LIN {X 0,Y 523.947,Z 221.718,A -85,B 0,C 180,E1 -4737.68,E2 -4737.68} C_VEL
LIN {X 0,Y 523.963,Z 221.716,A -85,B 0,C 180,E1 -4740.677,E2 -4740.677} C_VEL
LIN {X 0,Y 523.944,Z 221.72,A -85,B 0,C 180,E1 -4743.726,E2 -4743.726} C_VEL
LIN {X 0,Y 523.98,Z 221.866,A -85,B 0,C 180,E1 -4746.586,E2 -4746.586} C_VEL
LIN {X 0,Y 525.206,Z 229.619,A -85,B 0,C 180,E1 -4747.994,E2 -4747.994} C_VEL
LIN {X 0,Y 524.786,Z 247.778,A -85,B 0,C 180,E1 -4751.048,E2 -4751.048} C_VEL
LIN {X 0,Y 524.374,Z 265.93,A -85,B 0,C 180,E1 -4754.052,E2 -4754.052} C_VEL
LIN {X 0,Y 524.311,Z 270.834,A -85,B 0,C 180,E1 -4754.823,E2 -4754.823} C_VEL
LIN {X 0,Y 525.641,Z 279.389,A -85,B 0,C 180,E1 -4755.009,E2 -4755.009} C_VEL
LIN {X 0,Y 525.957,Z 285.477,A -85,B 0,C 180,E1 -4755.103,E2 -4755.103} C_VEL
LIN {X 0,Y 525.554,Z 378.201,A -85,B 0,C 180,E1 -4756.391,E2 -4756.391} C_VEL
LIN {X 0,Y 525.355,Z 391.598,A -85,B 0,C 180,E1 -4756.731,E2 -4756.731} C_VEL
LIN {X 0,Y 525.029,Z 404.942,A -85,B 0,C 180,E1 -4757.239,E2 -4757.239} C_VEL
LIN {X 0,Y 524.818,Z 416.473,A -85,B 0,C 180,E1 -4757.844,E2 -4757.844} C_VEL
LIN {X 0,Y 524.548,Z 427.744,A -85,B 0,C 180,E1 -4758.601,E2 -4758.601} C_VEL
LIN {X 0,Y 524.212,Z 438.191,A -85,B 0,C 180,E1 -4759.474,E2 -4759.474} C_VEL
LIN {X 0,Y 524.028,Z 446.732,A -85,B 0,C 180,E1 -4760.348,E2 -4760.348} C_VEL
LIN {X 0,Y 523.819,Z 454.609,A -85,B 0,C 180,E1 -4761.317,E2 -4761.317} C_VEL
LIN {X 0,Y 523.624,Z 462.299,A -85,B 0,C 180,E1 -4762.479,E2 -4762.479} C_VEL
LIN {X 0,Y 523.496,Z 469.383,A -85,B 0,C 180,E1 -4763.833,E2 -4763.833} C_VEL
LIN {X 0,Y 523.385,Z 474.095,A -85,B 0,C 180,E1 -4764.992,E2 -4764.992} C_VEL
LIN {X 0,Y 523.445,Z 477.695,A -85,B 0,C 180,E1 -4766.15,E2 -4766.15} C_VEL
LIN {X 0,Y 523.369,Z 479.552,A -85,B 0,C 180,E1 -4766.92,E2 -4766.92} C_VEL
LIN {X 0,Y 523.335,Z 480.943,A -85,B 0,C 180,E1 -4767.69,E2 -4767.69} C_VEL
LIN {X 0,Y 523.25,Z 482.542,A -85,B 0,C 180,E1 -4769.229,E2 -4769.229} C_VEL
LIN {X 0,Y 523.247,Z 482.758,A -85,B 0,C 180,E1 -4769.999,E2 -4769.999} C_VEL
LIN {X 0,Y 523.275,Z 481.938,A -85,B 0,C 180,E1 -4771.538,E2 -4771.538} C_VEL
LIN {X 0,Y 523.335,Z 480.947,A -85,B 0,C 180,E1 -4772.308,E2 -4772.308} C_VEL
LIN {X 0,Y 523.368,Z 479.556,A -85,B 0,C 180,E1 -4773.078,E2 -4773.078} C_VEL
LIN {X 0,Y 523.424,Z 476.63,A -85,B 0,C 180,E1 -4774.234,E2 -4774.234} C_VEL
LIN {X 0,Y 523.462,Z 472.668,A -85,B 0,C 180,E1 -4775.391,E2 -4775.391} C_VEL
LIN {X 0,Y 523.503,Z 466.604,A -85,B 0,C 180,E1 -4776.738,E2 -4776.738} C_VEL
LIN {X 0,Y 523.674,Z 459.908,A -85,B 0,C 180,E1 -4777.905,E2 -4777.905} C_VEL
LIN {X 0,Y 523.861,Z 451.635,A -85,B 0,C 180,E1 -4779.068,E2 -4779.068} C_VEL
LIN {X 0,Y 524.081,Z 443.153,A -85,B 0,C 180,E1 -4780.038,E2 -4780.038} C_VEL
LIN {X 0,Y 524.365,Z 432.668,A -85,B 0,C 180,E1 -4781.009,E2 -4781.009} C_VEL
LIN {X 0,Y 524.659,Z 421.21,A -85,B 0,C 180,E1 -4781.86,E2 -4781.86} C_VEL
LIN {X 0,Y 524.974,Z 408.979,A -85,B 0,C 180,E1 -4782.563,E2 -4782.563} C_VEL
LIN {X 0,Y 525.247,Z 396.61,A -85,B 0,C 180,E1 -4783.097,E2 -4783.097} C_VEL
LIN {X 0,Y 525.41,Z 383.894,A -85,B 0,C 180,E1 -4783.487,E2 -4783.487} C_VEL
LIN {X 0,Y 525.622,Z 368.754,A -85,B 0,C 180,E1 -4783.752,E2 -4783.752} C_VEL
LIN {X 0,Y 525.857,Z 280.922,A -85,B 0,C 180,E1 -4784.963,E2 -4784.963} C_VEL
LIN {X 0,Y 524.29,Z 270.905,A -85,B 0,C 180,E1 -4785.169,E2 -4785.169} C_VEL
LIN {X 0,Y 524.336,Z 265.85,A -85,B 0,C 180,E1 -4785.947,E2 -4785.947} C_VEL
LIN {X 0,Y 524.686,Z 248.802,A -85,B 0,C 180,E1 -4788.751,E2 -4788.751} C_VEL
LIN {X 0,Y 525.189,Z 230.523,A -85,B 0,C 180,E1 -4791.797,E2 -4791.797} C_VEL
LIN {X 0,Y 524.722,Z 225.824,A -85,B 0,C 180,E1 -4792.615,E2 -4792.615} C_VEL
LIN {X 0,Y 523.962,Z 221.786,A -85,B 0,C 180,E1 -4793.386,E2 -4793.386} C_VEL
LIN {X 0,Y 523.944,Z 221.72,A -85,B 0,C 180,E1 -4796.272,E2 -4796.272} C_VEL
LIN {X 0,Y 523.931,Z 221.717,A -85,B 0,C 180,E1 -4798.874,E2 -4798.874} C_VEL
LIN {X 0,Y 523.921,Z 221.723,A -85,B 0,C 180,E1 -4801.542,E2 -4801.542} C_VEL
LIN {X 0,Y 523.932,Z 221.72,A -85,B 0,C 180,E1 -4804.288,E2 -4804.288} C_VEL
LIN {X 0,Y 523.904,Z 221.721,A -85,B 0,C 180,E1 -4807.131,E2 -4807.131} C_VEL
LIN {X 0,Y 523.938,Z 221.725,A -85,B 0,C 180,E1 -4810.128,E2 -4810.128} C_VEL
LIN {X 0,Y 523.922,Z 221.723,A -85,B 0,C 180,E1 -4812.455,E2 -4812.455} C_VEL
LIN {X 0,Y 523.94,Z 221.715,A -85,B 0,C 180,E1 -4815.308,E2 -4815.308} C_VEL
LIN {X 0,Y 523.938,Z 221.721,A -85,B 0,C 180,E1 -4818.69,E2 -4818.69} C_VEL
LIN {X 0,Y 523.909,Z 221.721,A -85,B 0,C 180,E1 -4821.896,E2 -4821.896} C_VEL
LIN {X 0,Y 523.919,Z 221.722,A -85,B 0,C 180,E1 -4824.909,E2 -4824.909} C_VEL
LIN {X 0,Y 523.93,Z 221.715,A -85,B 0,C 180,E1 -4827.678,E2 -4827.678} C_VEL
LIN {X 0,Y 523.946,Z 221.722,A -85,B 0,C 180,E1 -4830.675,E2 -4830.675} C_VEL
LIN {X 0,Y 523.898,Z 221.72,A -85,B 0,C 180,E1 -4833.722,E2 -4833.722} C_VEL
LIN {X 0,Y 523.9,Z 221.721,A -85,B 0,C 180,E1 -4836.267,E2 -4836.267} C_VEL
LIN {X 0,Y 523.935,Z 221.722,A -85,B 0,C 180,E1 -4838.764,E2 -4838.764} C_VEL
LIN {X 0,Y 523.928,Z 221.723,A -85,B 0,C 180,E1 -4841.217,E2 -4841.217} C_VEL
LIN {X 0,Y 523.899,Z 221.721,A -85,B 0,C 180,E1 -4843.635,E2 -4843.635} C_VEL
LIN {X 0,Y 523.902,Z 221.72,A -85,B 0,C 180,E1 -4846.024,E2 -4846.024} C_VEL
LIN {X 0,Y 524.003,Z 221.705,A -85,B 0,C 180,E1 -4848.391,E2 -4848.391} C_VEL
LIN {X 0,Y 523.934,Z 221.719,A -85,B 0,C 180,E1 -4851.512,E2 -4851.512} C_VEL
LIN {X 0,Y 523.997,Z 221.711,A -85,B 0,C 180,E1 -4853.838,E2 -4853.838} C_VEL
LIN {X 0,Y 523.934,Z 221.725,A -85,B 0,C 180,E1 -4855.381,E2 -4855.381} C_VEL
LIN {X 0,Y 524.082,Z 221.703,A -85,B 0,C 180,E1 -4857.691,E2 -4857.691} C_VEL
LIN {X 0,Y 524.071,Z 221.7,A -85,B 0,C 180,E1 -4859.997,E2 -4859.997} C_VEL
LIN {X 0,Y 524.079,Z 221.698,A -85,B 0,C 180,E1 -4862.303,E2 -4862.303} C_VEL
LIN {X 0,Y 523.982,Z 221.713,A -85,B 0,C 180,E1 -4866.157,E2 -4866.157} C_VEL
LIN {X 0,Y 523.96,Z 221.714,A -85,B 0,C 180,E1 -4869.259,E2 -4869.259} C_VEL
LIN {X 0,Y 523.977,Z 221.719,A -85,B 0,C 180,E1 -4871.734,E2 -4871.734} C_VEL
LIN {X 0,Y 523.963,Z 221.713,A -85,B 0,C 180,E1 -4875.046,E2 -4875.046} C_VEL
LIN {X 0,Y 523.92,Z 221.726,A -85,B 0,C 180,E1 -4877.967,E2 -4877.967} C_VEL
LIN {X 0,Y 523.946,Z 221.72,A -85,B 0,C 180,E1 -4880.407,E2 -4880.407} C_VEL
LIN {X 0,Y 523.884,Z 221.723,A -85,B 0,C 180,E1 -4882.891,E2 -4882.891} C_VEL
LIN {X 0,Y 523.954,Z 221.719,A -85,B 0,C 180,E1 -4886.016,E2 -4886.016} C_VEL
LIN {X 0,Y 523.908,Z 221.72,A -85,B 0,C 180,E1 -4888.872,E2 -4888.872} C_VEL
LIN {X 0,Y 523.891,Z 221.722,A -85,B 0,C 180,E1 -4891.541,E2 -4891.541} C_VEL
LIN {X 0,Y 523.912,Z 221.726,A -85,B 0,C 180,E1 -4894.287,E2 -4894.287} C_VEL
LIN {X 0,Y 523.879,Z 221.726,A -85,B 0,C 180,E1 -4897.129,E2 -4897.129} C_VEL
LIN {X 0,Y 523.932,Z 221.72,A -85,B 0,C 180,E1 -4900.132,E2 -4900.132} C_VEL
LIN {X 0,Y 523.908,Z 221.726,A -85,B 0,C 180,E1 -4902.458,E2 -4902.458} C_VEL
LIN {X 0,Y 523.917,Z 221.724,A -85,B 0,C 180,E1 -4905.306,E2 -4905.306} C_VEL
LIN {X 0,Y 523.893,Z 221.73,A -85,B 0,C 180,E1 -4906.862,E2 -4906.862} C_VEL
LIN {X 0,Y 523.611,Z 222.17,A -85,B 0,C 180,E1 -4907.286,E2 -4907.286} C_VEL
LIN {X 0,Y 522.901,Z 223.307,A -85,B 0,C 180,E1 -4907.69,E2 -4907.69} C_VEL
LIN {X 0,Y 520.809,Z 226.879,A -85,B 0,C 180,E1 -4908.44,E2 -4908.44} C_VEL
LIN {X 0,Y 518.658,Z 231.406,A -85,B 0,C 180,E1 -4909.162,E2 -4909.162} C_VEL
LIN {X 0,Y 517.705,Z 234.729,A -85,B 0,C 180,E1 -4909.714,E2 -4909.714} C_VEL
LIN {X 0,Y 517.612,Z 235.807,A -85,B 0,C 180,E1 -4909.904,E2 -4909.904} C_VEL
LIN {X 0,Y 517.285,Z 252.208,A -85,B 0,C 180,E1 -4912.803,E2 -4912.803} C_VEL
LIN {X 0,Y 517.261,Z 257.358,A -85,B 0,C 180,E1 -4913.666,E2 -4913.666} C_VEL
LIN {X 0,Y 519.08,Z 267.962,A -85,B 0,C 180,E1 -4913.896,E2 -4913.896} C_VEL
LIN {X 0,Y 518.62,Z 364.773,A -85,B 0,C 180,E1 -4915.266,E2 -4915.266} C_VEL
LIN {X 0,Y 518.388,Z 378.478,A -85,B 0,C 180,E1 -4915.628,E2 -4915.628} C_VEL
LIN {X 0,Y 518.17,Z 391.423,A -85,B 0,C 180,E1 -4916.141,E2 -4916.141} C_VEL
LIN {X 0,Y 517.873,Z 403.178,A -85,B 0,C 180,E1 -4916.777,E2 -4916.777} C_VEL
LIN {X 0,Y 517.535,Z 414.859,A -85,B 0,C 180,E1 -4917.588,E2 -4917.588} C_VEL
LIN {X 0,Y 517.253,Z 424.904,A -85,B 0,C 180,E1 -4918.461,E2 -4918.461} C_VEL
LIN {X 0,Y 516.989,Z 433.313,A -85,B 0,C 180,E1 -4919.353,E2 -4919.353} C_VEL
LIN {X 0,Y 516.714,Z 442.175,A -85,B 0,C 180,E1 -4920.505,E2 -4920.505} C_VEL
LIN {X 0,Y 516.594,Z 448.832,A -85,B 0,C 180,E1 -4921.567,E2 -4921.567} C_VEL
LIN {X 0,Y 516.445,Z 455.453,A -85,B 0,C 180,E1 -4922.88,E2 -4922.88} C_VEL
LIN {X 0,Y 516.342,Z 460.483,A -85,B 0,C 180,E1 -4924.181,E2 -4924.181} C_VEL
LIN {X 0,Y 516.281,Z 463.056,A -85,B 0,C 180,E1 -4925.041,E2 -4925.041} C_VEL
LIN {X 0,Y 516.233,Z 465.12,A -85,B 0,C 180,E1 -4925.896,E2 -4925.896} C_VEL
LIN {X 0,Y 516.168,Z 466.619,A -85,B 0,C 180,E1 -4926.745,E2 -4926.745} C_VEL
LIN {X 0,Y 516.15,Z 467.852,A -85,B 0,C 180,E1 -4927.791,E2 -4927.791} C_VEL
LIN {X 0,Y 516.16,Z 468.321,A -85,B 0,C 180,E1 -4929.268,E2 -4929.268} C_VEL
LIN {X 0,Y 516.202,Z 467.974,A -85,B 0,C 180,E1 -4930.102,E2 -4930.102} C_VEL
LIN {X 0,Y 516.163,Z 467.205,A -85,B 0,C 180,E1 -4930.928,E2 -4930.928} C_VEL
LIN {X 0,Y 516.222,Z 464.765,A -85,B 0,C 180,E1 -4932.347,E2 -4932.347} C_VEL
LIN {X 0,Y 516.313,Z 460.827,A -85,B 0,C 180,E1 -4933.798,E2 -4933.798} C_VEL
LIN {X 0,Y 516.425,Z 456.142,A -85,B 0,C 180,E1 -4935.048,E2 -4935.048} C_VEL
LIN {X 0,Y 516.564,Z 449.361,A -85,B 0,C 180,E1 -4936.428,E2 -4936.428} C_VEL
LIN {X 0,Y 516.761,Z 441.828,A -85,B 0,C 180,E1 -4937.633,E2 -4937.633} C_VEL
LIN {X 0,Y 516.945,Z 434.081,A -85,B 0,C 180,E1 -4938.643,E2 -4938.643} C_VEL
LIN {X 0,Y 517.271,Z 424.866,A -85,B 0,C 180,E1 -4939.63,E2 -4939.63} C_VEL
LIN {X 0,Y 517.531,Z 414.551,A -85,B 0,C 180,E1 -4940.524,E2 -4940.524} C_VEL
LIN {X 0,Y 517.896,Z 403.064,A -85,B 0,C 180,E1 -4941.318,E2 -4941.318} C_VEL
LIN {X 0,Y 518.131,Z 391.865,A -85,B 0,C 180,E1 -4941.927,E2 -4941.927} C_VEL
LIN {X 0,Y 518.4,Z 379.448,A -85,B 0,C 180,E1 -4942.43,E2 -4942.43} C_VEL
LIN {X 0,Y 518.63,Z 366.936,A -85,B 0,C 180,E1 -4942.776,E2 -4942.776} C_VEL
LIN {X 0,Y 518.731,Z 346.658,A -85,B 0,C 180,E1 -4943.095,E2 -4943.095} C_VEL
LIN {X 0,Y 518.965,Z 267.136,A -85,B 0,C 180,E1 -4944.208,E2 -4944.208} C_VEL
LIN {X 0,Y 517.256,Z 257.525,A -85,B 0,C 180,E1 -4944.421,E2 -4944.421} C_VEL
LIN {X 0,Y 517.473,Z 246.928,A -85,B 0,C 180,E1 -4946.302,E2 -4946.302} C_VEL
LIN {X 0,Y 517.903,Z 232.103,A -85,B 0,C 180,E1 -4949.029,E2 -4949.029} C_VEL
LIN {X 0,Y 517.75,Z 226.931,A -85,B 0,C 180,E1 -4950.001,E2 -4950.001} C_VEL
LIN {X 0,Y 517.036,Z 222.663,A -85,B 0,C 180,E1 -4950.877,E2 -4950.877} C_VEL
LIN {X 0,Y 516.976,Z 222.591,A -85,B 0,C 180,E1 -4953.118,E2 -4953.118} C_VEL
LIN {X 0,Y 516.961,Z 222.586,A -85,B 0,C 180,E1 -4956.245,E2 -4956.245} C_VEL
LIN {X 0,Y 516.909,Z 222.598,A -85,B 0,C 180,E1 -4959.391,E2 -4959.391} C_VEL
LIN {X 0,Y 516.941,Z 222.593,A -85,B 0,C 180,E1 -4961.826,E2 -4961.826} C_VEL
LIN {X 0,Y 516.901,Z 222.593,A -85,B 0,C 180,E1 -4965.148,E2 -4965.148} C_VEL
LIN {X 0,Y 516.884,Z 222.597,A -85,B 0,C 180,E1 -4968.225,E2 -4968.225} C_VEL
LIN {X 0,Y 516.873,Z 222.595,A -85,B 0,C 180,E1 -4970.704,E2 -4970.704} C_VEL
LIN {X 0,Y 516.851,Z 222.607,A -85,B 0,C 180,E1 -4974.076,E2 -4974.076} C_VEL
LIN {X 0,Y 516.851,Z 222.6,A -85,B 0,C 180,E1 -4976.663,E2 -4976.663} C_VEL
LIN {X 0,Y 516.875,Z 222.596,A -85,B 0,C 180,E1 -4979.527,E2 -4979.527} C_VEL
LIN {X 0,Y 516.861,Z 222.602,A -85,B 0,C 180,E1 -4982.546,E2 -4982.546} C_VEL
LIN {X 0,Y 516.821,Z 222.601,A -85,B 0,C 180,E1 -4985.331,E2 -4985.331} C_VEL
LIN {X 0,Y 516.843,Z 222.605,A -85,B 0,C 180,E1 -4988.72,E2 -4988.72} C_VEL
LIN {X 0,Y 516.854,Z 222.598,A -85,B 0,C 180,E1 -4991.782,E2 -4991.782} C_VEL
LIN {X 0,Y 516.871,Z 222.6,A -85,B 0,C 180,E1 -4995.011,E2 -4995.011} C_VEL
LIN {X 0,Y 516.865,Z 222.6,A -85,B 0,C 180,E1 -4998.406,E2 -4998.406} C_VEL
LIN {X 0,Y 516.856,Z 222.601,A -85,B 0,C 180,E1 -5001.288,E2 -5001.288} C_VEL
LIN {X 0,Y 516.853,Z 222.598,A -85,B 0,C 180,E1 -5004.224,E2 -5004.224} C_VEL
LIN {X 0,Y 516.864,Z 222.606,A -85,B 0,C 180,E1 -5007.056,E2 -5007.056} C_VEL
LIN {X 0,Y 516.849,Z 222.599,A -85,B 0,C 180,E1 -5009.798,E2 -5009.798} C_VEL
LIN {X 0,Y 516.861,Z 222.597,A -85,B 0,C 180,E1 -5012.468,E2 -5012.468} C_VEL
LIN {X 0,Y 516.861,Z 222.602,A -85,B 0,C 180,E1 -5015.65,E2 -5015.65} C_VEL
LIN {X 0,Y 516.878,Z 222.594,A -85,B 0,C 180,E1 -5018.466,E2 -5018.466} C_VEL
LIN {X 0,Y 516.884,Z 222.595,A -85,B 0,C 180,E1 -5020.958,E2 -5020.958} C_VEL
LIN {X 0,Y 516.878,Z 222.601,A -85,B 0,C 180,E1 -5023.413,E2 -5023.413} C_VEL
LIN {X 0,Y 516.879,Z 222.602,A -85,B 0,C 180,E1 -5025.837,E2 -5025.837} C_VEL
LIN {X 0,Y 516.926,Z 222.591,A -85,B 0,C 180,E1 -5028.236,E2 -5028.236} C_VEL
LIN {X 0,Y 516.93,Z 222.591,A -85,B 0,C 180,E1 -5031.402,E2 -5031.402} C_VEL
LIN {X 0,Y 516.983,Z 222.583,A -85,B 0,C 180,E1 -5034.543,E2 -5034.543} C_VEL
LIN {X 0,Y 517.075,Z 222.573,A -85,B 0,C 180,E1 -5037.666,E2 -5037.666} C_VEL
LIN {X 0,Y 517.072,Z 222.572,A -85,B 0,C 180,E1 -5040.782,E2 -5040.782} C_VEL
LIN {X 0,Y 516.949,Z 222.586,A -85,B 0,C 180,E1 -5043.12,E2 -5043.12} C_VEL
LIN {X 0,Y 516.978,Z 222.59,A -85,B 0,C 180,E1 -5046.246,E2 -5046.246} C_VEL
LIN {X 0,Y 516.918,Z 222.589,A -85,B 0,C 180,E1 -5049.393,E2 -5049.393} C_VEL
LIN {X 0,Y 516.964,Z 222.584,A -85,B 0,C 180,E1 -5051.809,E2 -5051.809} C_VEL
LIN {X 0,Y 516.949,Z 222.588,A -85,B 0,C 180,E1 -5055.145,E2 -5055.145} C_VEL
LIN {X 0,Y 516.923,Z 222.591,A -85,B 0,C 180,E1 -5058.225,E2 -5058.225} C_VEL
LIN {X 0,Y 516.914,Z 222.598,A -85,B 0,C 180,E1 -5060.704,E2 -5060.704} C_VEL
LIN {X 0,Y 516.869,Z 222.6,A -85,B 0,C 180,E1 -5063.226,E2 -5063.226} C_VEL
LIN {X 0,Y 516.895,Z 222.592,A -85,B 0,C 180,E1 -5066.183,E2 -5066.183} C_VEL
LIN {X 0,Y 516.917,Z 222.596,A -85,B 0,C 180,E1 -5069.307,E2 -5069.307} C_VEL
LIN {X 0,Y 516.905,Z 222.592,A -85,B 0,C 180,E1 -5072.543,E2 -5072.543} C_VEL
LIN {X 0,Y 516.868,Z 222.606,A -85,B 0,C 180,E1 -5075.328,E2 -5075.328} C_VEL
LIN {X 0,Y 516.891,Z 222.595,A -85,B 0,C 180,E1 -5077.943,E2 -5077.943} C_VEL
LIN {X 0,Y 516.866,Z 222.596,A -85,B 0,C 180,E1 -5080.745,E2 -5080.745} C_VEL
LIN {X 0,Y 516.894,Z 222.597,A -85,B 0,C 180,E1 -5083.904,E2 -5083.904} C_VEL
LIN {X 0,Y 516.893,Z 222.596,A -85,B 0,C 180,E1 -5086.108,E2 -5086.108} C_VEL
LIN {X 0,Y 516.865,Z 222.598,A -85,B 0,C 180,E1 -5089.255,E2 -5089.255} C_VEL
LIN {X 0,Y 516.873,Z 222.599,A -85,B 0,C 180,E1 -5092.274,E2 -5092.274} C_VEL
LIN {X 0,Y 516.892,Z 222.593,A -85,B 0,C 180,E1 -5095.175,E2 -5095.175} C_VEL
LIN {X 0,Y 516.885,Z 222.602,A -85,B 0,C 180,E1 -5097.975,E2 -5097.975} C_VEL
LIN {X 0,Y 516.931,Z 222.592,A -85,B 0,C 180,E1 -5100.695,E2 -5100.695} C_VEL
LIN {X 0,Y 516.909,Z 222.597,A -85,B 0,C 180,E1 -5103.814,E2 -5103.814} C_VEL
LIN {X 0,Y 516.941,Z 222.705,A -85,B 0,C 180,E1 -5106.407,E2 -5106.407} C_VEL
LIN {X 0,Y 518.254,Z 230.732,A -85,B 0,C 180,E1 -5107.893,E2 -5107.893} C_VEL
LIN {X 0,Y 517.84,Z 247.689,A -85,B 0,C 180,E1 -5110.784,E2 -5110.784} C_VEL
LIN {X 0,Y 517.378,Z 265.836,A -85,B 0,C 180,E1 -5113.83,E2 -5113.83} C_VEL
LIN {X 0,Y 517.302,Z 270.899,A -85,B 0,C 180,E1 -5114.622,E2 -5114.622} C_VEL
LIN {X 0,Y 519.108,Z 283.14,A -85,B 0,C 180,E1 -5114.87,E2 -5114.87} C_VEL
LIN {X 0,Y 518.659,Z 378.034,A -85,B 0,C 180,E1 -5116.207,E2 -5116.207} C_VEL
LIN {X 0,Y 518.443,Z 391.457,A -85,B 0,C 180,E1 -5116.55,E2 -5116.55} C_VEL
LIN {X 0,Y 518.082,Z 404.812,A -85,B 0,C 180,E1 -5117.065,E2 -5117.065} C_VEL
LIN {X 0,Y 517.838,Z 417.3,A -85,B 0,C 180,E1 -5117.737,E2 -5117.737} C_VEL
LIN {X 0,Y 517.529,Z 428.922,A -85,B 0,C 180,E1 -5118.543,E2 -5118.543} C_VEL
LIN {X 0,Y 517.166,Z 439.128,A -85,B 0,C 180,E1 -5119.428,E2 -5119.428} C_VEL
LIN {X 0,Y 516.948,Z 448.304,A -85,B 0,C 180,E1 -5120.412,E2 -5120.412} C_VEL
LIN {X 0,Y 516.696,Z 457.24,A -85,B 0,C 180,E1 -5121.591,E2 -5121.591} C_VEL
LIN {X 0,Y 516.51,Z 464.43,A -85,B 0,C 180,E1 -5122.768,E2 -5122.768} C_VEL
LIN {X 0,Y 516.426,Z 470.976,A -85,B 0,C 180,E1 -5124.141,E2 -5124.141} C_VEL
LIN {X 0,Y 516.27,Z 475.304,A -85,B 0,C 180,E1 -5125.314,E2 -5125.314} C_VEL
LIN {X 0,Y 516.354,Z 477.596,A -85,B 0,C 180,E1 -5126.097,E2 -5126.097} C_VEL
LIN {X 0,Y 516.284,Z 479.453,A -85,B 0,C 180,E1 -5126.877,E2 -5126.877} C_VEL
LIN {X 0,Y 516.262,Z 480.845,A -85,B 0,C 180,E1 -5127.658,E2 -5127.658} C_VEL
LIN {X 0,Y 516.161,Z 482.443,A -85,B 0,C 180,E1 -5129.219,E2 -5129.219} C_VEL
LIN {X 0,Y 516.155,Z 482.66,A -85,B 0,C 180,E1 -5129.999,E2 -5129.999} C_VEL
LIN {X 0,Y 516.192,Z 481.84,A -85,B 0,C 180,E1 -5131.559,E2 -5131.559} C_VEL
LIN {X 0,Y 516.261,Z 480.848,A -85,B 0,C 180,E1 -5132.339,E2 -5132.339} C_VEL
LIN {X 0,Y 516.283,Z 479.456,A -85,B 0,C 180,E1 -5133.12,E2 -5133.12} C_VEL
LIN {X 0,Y 516.313,Z 476.529,A -85,B 0,C 180,E1 -5134.292,E2 -5134.292} C_VEL
LIN {X 0,Y 516.398,Z 472.565,A -85,B 0,C 180,E1 -5135.465,E2 -5135.465} C_VEL
LIN {X 0,Y 516.421,Z 467.366,A -85,B 0,C 180,E1 -5136.661,E2 -5136.661} C_VEL
LIN {X 0,Y 516.583,Z 461.034,A -85,B 0,C 180,E1 -5137.818,E2 -5137.818} C_VEL
LIN {X 0,Y 516.771,Z 453.014,A -85,B 0,C 180,E1 -5138.997,E2 -5138.997} C_VEL
LIN {X 0,Y 517.025,Z 444.838,A -85,B 0,C 180,E1 -5139.979,E2 -5139.979} C_VEL
LIN {X 0,Y 517.333,Z 434.866,A -85,B 0,C 180,E1 -5140.963,E2 -5140.963} C_VEL
LIN {X 0,Y 517.654,Z 424.006,A -85,B 0,C 180,E1 -5141.82,E2 -5141.82} C_VEL
LIN {X 0,Y 517.955,Z 412.551,A -85,B 0,C 180,E1 -5142.537,E2 -5142.537} C_VEL
LIN {X 0,Y 518.226,Z 400.301,A -85,B 0,C 180,E1 -5143.128,E2 -5143.128} C_VEL
LIN {X 0,Y 518.452,Z 387.398,A -85,B 0,C 180,E1 -5143.572,E2 -5143.572} C_VEL
LIN {X 0,Y 518.682,Z 373.677,A -85,B 0,C 180,E1 -5143.865,E2 -5143.865} C_VEL
LIN {X 0,Y 518.981,Z 281.581,A -85,B 0,C 180,E1 -5145.155,E2 -5145.155} C_VEL
LIN {X 0,Y 517.258,Z 270.805,A -85,B 0,C 180,E1 -5145.38,E2 -5145.38} C_VEL
LIN {X 0,Y 517.458,Z 260.873,A -85,B 0,C 180,E1 -5146.977,E2 -5146.977} C_VEL
LIN {X 0,Y 517.817,Z 245.05,A -85,B 0,C 180,E1 -5149.627,E2 -5149.627} C_VEL
LIN {X 0,Y 518.236,Z 230.421,A -85,B 0,C 180,E1 -5152.105,E2 -5152.105} C_VEL
LIN {X 0,Y 516.929,Z 222.695,A -85,B 0,C 180,E1 -5153.537,E2 -5153.537} C_VEL
LIN {X 0,Y 516.912,Z 222.594,A -85,B 0,C 180,E1 -5156.657,E2 -5156.657} C_VEL
LIN {X 0,Y 516.91,Z 222.597,A -85,B 0,C 180,E1 -5159.521,E2 -5159.521} C_VEL
LIN {X 0,Y 516.897,Z 222.594,A -85,B 0,C 180,E1 -5162.541,E2 -5162.541} C_VEL
LIN {X 0,Y 516.864,Z 222.597,A -85,B 0,C 180,E1 -5165.327,E2 -5165.327} C_VEL
LIN {X 0,Y 516.878,Z 222.601,A -85,B 0,C 180,E1 -5167.941,E2 -5167.941} C_VEL
LIN {X 0,Y 516.881,Z 222.596,A -85,B 0,C 180,E1 -5170.74,E2 -5170.74} C_VEL
LIN {X 0,Y 516.88,Z 222.599,A -85,B 0,C 180,E1 -5173.901,E2 -5173.901} C_VEL
LIN {X 0,Y 516.88,Z 222.599,A -85,B 0,C 180,E1 -5176.105,E2 -5176.105} C_VEL
LIN {X 0,Y 516.901,Z 222.6,A -85,B 0,C 180,E1 -5178.398,E2 -5178.398} C_VEL
LIN {X 0,Y 516.873,Z 222.596,A -85,B 0,C 180,E1 -5181.281,E2 -5181.281} C_VEL
LIN {X 0,Y 516.864,Z 222.601,A -85,B 0,C 180,E1 -5184.217,E2 -5184.217} C_VEL
LIN {X 0,Y 516.891,Z 222.595,A -85,B 0,C 180,E1 -5187.051,E2 -5187.051} C_VEL
LIN {X 0,Y 516.877,Z 222.595,A -85,B 0,C 180,E1 -5189.793,E2 -5189.793} C_VEL
LIN {X 0,Y 516.885,Z 222.599,A -85,B 0,C 180,E1 -5192.463,E2 -5192.463} C_VEL
LIN {X 0,Y 516.865,Z 222.596,A -85,B 0,C 180,E1 -5195.643,E2 -5195.643} C_VEL
LIN {X 0,Y 516.876,Z 222.597,A -85,B 0,C 180,E1 -5198.459,E2 -5198.459} C_VEL
LIN {X 0,Y 516.881,Z 222.603,A -85,B 0,C 180,E1 -5200.952,E2 -5200.952} C_VEL
LIN {X 0,Y 516.879,Z 222.598,A -85,B 0,C 180,E1 -5203.407,E2 -5203.407} C_VEL
LIN {X 0,Y 516.861,Z 222.598,A -85,B 0,C 180,E1 -5205.83,E2 -5205.83} C_VEL
LIN {X 0,Y 516.931,Z 222.592,A -85,B 0,C 180,E1 -5209.025,E2 -5209.025} C_VEL
LIN {X 0,Y 516.928,Z 222.585,A -85,B 0,C 180,E1 -5212.183,E2 -5212.183} C_VEL
LIN {X 0,Y 516.998,Z 222.58,A -85,B 0,C 180,E1 -5214.537,E2 -5214.537} C_VEL
LIN {X 0,Y 517.053,Z 222.58,A -85,B 0,C 180,E1 -5217.66,E2 -5217.66} C_VEL
LIN {X 0,Y 517.041,Z 222.576,A -85,B 0,C 180,E1 -5219.997,E2 -5219.997} C_VEL
LIN {X 0,Y 517.05,Z 222.574,A -85,B 0,C 180,E1 -5222.334,E2 -5222.334} C_VEL
LIN {X 0,Y 516.949,Z 222.588,A -85,B 0,C 180,E1 -5226.241,E2 -5226.241} C_VEL
LIN {X 0,Y 516.916,Z 222.593,A -85,B 0,C 180,E1 -5229.386,E2 -5229.386} C_VEL
LIN {X 0,Y 516.931,Z 222.598,A -85,B 0,C 180,E1 -5231.804,E2 -5231.804} C_VEL
LIN {X 0,Y 516.916,Z 222.591,A -85,B 0,C 180,E1 -5235.141,E2 -5235.141} C_VEL
LIN {X 0,Y 516.887,Z 222.601,A -85,B 0,C 180,E1 -5238.22,E2 -5238.22} C_VEL
LIN {X 0,Y 516.886,Z 222.596,A -85,B 0,C 180,E1 -5240.698,E2 -5240.698} C_VEL
LIN {X 0,Y 516.863,Z 222.605,A -85,B 0,C 180,E1 -5244.07,E2 -5244.07} C_VEL
LIN {X 0,Y 516.894,Z 222.597,A -85,B 0,C 180,E1 -5246.655,E2 -5246.655} C_VEL
LIN {X 0,Y 516.88,Z 222.593,A -85,B 0,C 180,E1 -5249.521,E2 -5249.521} C_VEL
LIN {X 0,Y 516.865,Z 222.602,A -85,B 0,C 180,E1 -5252.541,E2 -5252.541} C_VEL
LIN {X 0,Y 516.85,Z 222.597,A -85,B 0,C 180,E1 -5255.33,E2 -5255.33} C_VEL
LIN {X 0,Y 516.848,Z 222.601,A -85,B 0,C 180,E1 -5257.941,E2 -5257.941} C_VEL
LIN {X 0,Y 516.872,Z 222.604,A -85,B 0,C 180,E1 -5260.737,E2 -5260.737} C_VEL
LIN {X 0,Y 516.845,Z 222.601,A -85,B 0,C 180,E1 -5263.901,E2 -5263.901} C_VEL
LIN {X 0,Y 516.845,Z 222.604,A -85,B 0,C 180,E1 -5266.105,E2 -5266.105} C_VEL
LIN {X 0,Y 516.93,Z 222.746,A -85,B 0,C 180,E1 -5267.517,E2 -5267.517} C_VEL
LIN {X 0,Y 517.73,Z 228.294,A -85,B 0,C 180,E1 -5268.57,E2 -5268.57} C_VEL
LIN {X 0,Y 517.612,Z 235.807,A -85,B 0,C 180,E1 -5269.904,E2 -5269.904} C_VEL
LIN {X 0,Y 516.894,Z 239.011,A -85,B 0,C 180,E1 -5270.447,E2 -5270.447} C_VEL
LIN {X 0,Y 511.014,Z 249.928,A -85,B 0,C 180,E1 -5272.178,E2 -5272.178} C_VEL
LIN {X 0,Y 510.295,Z 253.149,A -85,B 0,C 180,E1 -5272.731,E2 -5272.731} C_VEL
LIN {X 0,Y 510.251,Z 257.498,A -85,B 0,C 180,E1 -5273.452,E2 -5273.452} C_VEL
LIN {X 0,Y 512.263,Z 269.537,A -85,B 0,C 180,E1 -5273.711,E2 -5273.711} C_VEL
LIN {X 0,Y 511.751,Z 364.691,A -85,B 0,C 180,E1 -5275.075,E2 -5275.075} C_VEL
LIN {X 0,Y 511.523,Z 378.353,A -85,B 0,C 180,E1 -5275.438,E2 -5275.438} C_VEL
LIN {X 0,Y 511.28,Z 390.893,A -85,B 0,C 180,E1 -5275.936,E2 -5275.936} C_VEL
LIN {X 0,Y 510.996,Z 401.643,A -85,B 0,C 180,E1 -5276.507,E2 -5276.507} C_VEL
LIN {X 0,Y 510.652,Z 412.228,A -85,B 0,C 180,E1 -5277.22,E2 -5277.22} C_VEL
LIN {X 0,Y 510.334,Z 422.694,A -85,B 0,C 180,E1 -5278.099,E2 -5278.099} C_VEL
LIN {X 0,Y 510.011,Z 432.632,A -85,B 0,C 180,E1 -5279.13,E2 -5279.13} C_VEL
LIN {X 0,Y 509.73,Z 441.602,A -85,B 0,C 180,E1 -5280.289,E2 -5280.289} C_VEL
LIN {X 0,Y 509.523,Z 449.617,A -85,B 0,C 180,E1 -5281.586,E2 -5281.586} C_VEL
LIN {X 0,Y 509.372,Z 456.078,A -85,B 0,C 180,E1 -5282.917,E2 -5282.917} C_VEL
LIN {X 0,Y 509.248,Z 460.957,A -85,B 0,C 180,E1 -5284.234,E2 -5284.234} C_VEL
LIN {X 0,Y 509.156,Z 464.728,A -85,B 0,C 180,E1 -5285.633,E2 -5285.633} C_VEL
LIN {X 0,Y 509.091,Z 466.236,A -85,B 0,C 180,E1 -5286.402,E2 -5286.402} C_VEL
LIN {X 0,Y 509.065,Z 467.835,A -85,B 0,C 180,E1 -5287.652,E2 -5287.652} C_VEL
LIN {X 0,Y 509.048,Z 468.449,A -85,B 0,C 180,E1 -5288.965,E2 -5288.965} C_VEL
LIN {X 0,Y 509.102,Z 468.25,A -85,B 0,C 180,E1 -5289.823,E2 -5289.823} C_VEL
LIN {X 0,Y 509.094,Z 467.613,A -85,B 0,C 180,E1 -5290.653,E2 -5290.653} C_VEL
LIN {X 0,Y 509.087,Z 466.551,A -85,B 0,C 180,E1 -5291.489,E2 -5291.489} C_VEL
LIN {X 0,Y 509.14,Z 464.087,A -85,B 0,C 180,E1 -5292.737,E2 -5292.737} C_VEL
LIN {X 0,Y 509.246,Z 460.564,A -85,B 0,C 180,E1 -5293.979,E2 -5293.979} C_VEL
LIN {X 0,Y 509.37,Z 455.523,A -85,B 0,C 180,E1 -5295.299,E2 -5295.299} C_VEL
LIN {X 0,Y 509.499,Z 448.828,A -85,B 0,C 180,E1 -5296.643,E2 -5296.643} C_VEL
LIN {X 0,Y 509.721,Z 441.164,A -85,B 0,C 180,E1 -5297.863,E2 -5297.863} C_VEL
LIN {X 0,Y 509.977,Z 433.336,A -85,B 0,C 180,E1 -5298.877,E2 -5298.877} C_VEL
LIN {X 0,Y 510.295,Z 423.777,A -85,B 0,C 180,E1 -5299.888,E2 -5299.888} C_VEL
LIN {X 0,Y 510.608,Z 413.189,A -85,B 0,C 180,E1 -5300.794,E2 -5300.794} C_VEL
LIN {X 0,Y 510.998,Z 401.613,A -85,B 0,C 180,E1 -5301.583,E2 -5301.583} C_VEL
LIN {X 0,Y 511.311,Z 389.829,A -85,B 0,C 180,E1 -5302.2,E2 -5302.2} C_VEL
LIN {X 0,Y 511.562,Z 376.851,A -85,B 0,C 180,E1 -5302.7,E2 -5302.7} C_VEL
LIN {X 0,Y 511.789,Z 364.125,A -85,B 0,C 180,E1 -5303.026,E2 -5303.026} C_VEL
LIN {X 0,Y 512.123,Z 268.161,A -85,B 0,C 180,E1 -5304.402,E2 -5304.402} C_VEL
LIN {X 0,Y 510.297,Z 258.034,A -85,B 0,C 180,E1 -5304.618,E2 -5304.618} C_VEL
LIN {X 0,Y 510.235,Z 257.298,A -85,B 0,C 180,E1 -5304.667,E2 -5304.667} C_VEL
LIN {X 0,Y 510.696,Z 241.101,A -85,B 0,C 180,E1 -5307.635,E2 -5307.635} C_VEL
LIN {X 0,Y 510.926,Z 229.528,A -85,B 0,C 180,E1 -5309.804,E2 -5309.804} C_VEL
LIN {X 0,Y 509.982,Z 223.529,A -85,B 0,C 180,E1 -5311.038,E2 -5311.038} C_VEL
LIN {X 0,Y 509.919,Z 223.47,A -85,B 0,C 180,E1 -5313.162,E2 -5313.162} C_VEL
LIN {X 0,Y 509.912,Z 223.465,A -85,B 0,C 180,E1 -5316.332,E2 -5316.332} C_VEL
LIN {X 0,Y 509.872,Z 223.468,A -85,B 0,C 180,E1 -5318.722,E2 -5318.722} C_VEL
LIN {X 0,Y 509.909,Z 223.467,A -85,B 0,C 180,E1 -5321.933,E2 -5321.933} C_VEL
LIN {X 0,Y 509.853,Z 223.472,A -85,B 0,C 180,E1 -5325.244,E2 -5325.244} C_VEL
LIN {X 0,Y 509.848,Z 223.477,A -85,B 0,C 180,E1 -5328.003,E2 -5328.003} C_VEL
LIN {X 0,Y 509.811,Z 223.475,A -85,B 0,C 180,E1 -5331.005,E2 -5331.005} C_VEL
LIN {X 0,Y 509.783,Z 223.481,A -85,B 0,C 180,E1 -5333.567,E2 -5333.567} C_VEL
LIN {X 0,Y 509.816,Z 223.479,A -85,B 0,C 180,E1 -5336.368,E2 -5336.368} C_VEL
LIN {X 0,Y 509.815,Z 223.475,A -85,B 0,C 180,E1 -5338.849,E2 -5338.849} C_VEL
LIN {X 0,Y 509.786,Z 223.479,A -85,B 0,C 180,E1 -5341.594,E2 -5341.594} C_VEL
LIN {X 0,Y 509.801,Z 223.485,A -85,B 0,C 180,E1 -5344.418,E2 -5344.418} C_VEL
LIN {X 0,Y 509.761,Z 223.481,A -85,B 0,C 180,E1 -5347.347,E2 -5347.347} C_VEL
LIN {X 0,Y 509.785,Z 223.485,A -85,B 0,C 180,E1 -5350.388,E2 -5350.388} C_VEL
LIN {X 0,Y 509.769,Z 223.483,A -85,B 0,C 180,E1 -5353.063,E2 -5353.063} C_VEL
LIN {X 0,Y 509.798,Z 223.476,A -85,B 0,C 180,E1 -5355.797,E2 -5355.797} C_VEL
LIN {X 0,Y 509.809,Z 223.481,A -85,B 0,C 180,E1 -5358.576,E2 -5358.576} C_VEL
LIN {X 0,Y 509.83,Z 223.472,A -85,B 0,C 180,E1 -5361.791,E2 -5361.791} C_VEL
LIN {X 0,Y 509.811,Z 223.479,A -85,B 0,C 180,E1 -5364.626,E2 -5364.626} C_VEL
LIN {X 0,Y 509.842,Z 223.475,A -85,B 0,C 180,E1 -5367.485,E2 -5367.485} C_VEL
LIN {X 0,Y 509.84,Z 223.471,A -85,B 0,C 180,E1 -5370.279,E2 -5370.279} C_VEL
LIN {X 0,Y 509.808,Z 223.48,A -85,B 0,C 180,E1 -5372.945,E2 -5372.945} C_VEL
LIN {X 0,Y 509.823,Z 223.479,A -85,B 0,C 180,E1 -5375.576,E2 -5375.576} C_VEL
LIN {X 0,Y 509.814,Z 223.475,A -85,B 0,C 180,E1 -5378.152,E2 -5378.152} C_VEL
LIN {X 0,Y 509.85,Z 223.47,A -85,B 0,C 180,E1 -5380.685,E2 -5380.685} C_VEL
LIN {X 0,Y 509.847,Z 223.473,A -85,B 0,C 180,E1 -5383.177,E2 -5383.177} C_VEL
LIN {X 0,Y 509.85,Z 223.479,A -85,B 0,C 180,E1 -5385.637,E2 -5385.637} C_VEL
LIN {X 0,Y 509.889,Z 223.469,A -85,B 0,C 180,E1 -5388.134,E2 -5388.134} C_VEL
LIN {X 0,Y 509.884,Z 223.467,A -85,B 0,C 180,E1 -5391.283,E2 -5391.283} C_VEL
LIN {X 0,Y 509.918,Z 223.467,A -85,B 0,C 180,E1 -5393.673,E2 -5393.673} C_VEL
LIN {X 0,Y 509.892,Z 223.465,A -85,B 0,C 180,E1 -5396.843,E2 -5396.843} C_VEL
LIN {X 0,Y 509.932,Z 223.464,A -85,B 0,C 180,E1 -5398.424,E2 -5398.424} C_VEL
LIN {X 0,Y 510.023,Z 223.45,A -85,B 0,C 180,E1 -5400.793,E2 -5400.793} C_VEL
LIN {X 0,Y 510.045,Z 223.453,A -85,B 0,C 180,E1 -5402.372,E2 -5402.372} C_VEL
LIN {X 0,Y 509.947,Z 223.458,A -85,B 0,C 180,E1 -5405.539,E2 -5405.539} C_VEL
LIN {X 0,Y 509.883,Z 223.468,A -85,B 0,C 180,E1 -5407.925,E2 -5407.925} C_VEL
LIN {X 0,Y 509.917,Z 223.463,A -85,B 0,C 180,E1 -5411.128,E2 -5411.128} C_VEL
LIN {X 0,Y 509.859,Z 223.474,A -85,B 0,C 180,E1 -5414.369,E2 -5414.369} C_VEL
LIN {X 0,Y 509.875,Z 223.475,A -85,B 0,C 180,E1 -5416.828,E2 -5416.828} C_VEL
LIN {X 0,Y 509.92,Z 223.462,A -85,B 0,C 180,E1 -5420.158,E2 -5420.158} C_VEL
LIN {X 0,Y 509.831,Z 223.473,A -85,B 0,C 180,E1 -5423.566,E2 -5423.566} C_VEL
LIN {X 0,Y 509.831,Z 223.473,A -85,B 0,C 180,E1 -5426.358,E2 -5426.358} C_VEL
LIN {X 0,Y 509.85,Z 223.476,A -85,B 0,C 180,E1 -5428.848,E2 -5428.848} C_VEL
LIN {X 0,Y 509.826,Z 223.476,A -85,B 0,C 180,E1 -5431.592,E2 -5431.592} C_VEL
LIN {X 0,Y 509.847,Z 223.47,A -85,B 0,C 180,E1 -5434.416,E2 -5434.416} C_VEL
LIN {X 0,Y 509.82,Z 223.483,A -85,B 0,C 180,E1 -5437.343,E2 -5437.343} C_VEL
LIN {X 0,Y 509.827,Z 223.473,A -85,B 0,C 180,E1 -5440.385,E2 -5440.385} C_VEL
LIN {X 0,Y 509.82,Z 223.484,A -85,B 0,C 180,E1 -5443.574,E2 -5443.574} C_VEL
LIN {X 0,Y 509.819,Z 223.474,A -85,B 0,C 180,E1 -5446.427,E2 -5446.427} C_VEL
LIN {X 0,Y 509.827,Z 223.48,A -85,B 0,C 180,E1 -5449.616,E2 -5449.616} C_VEL
LIN {X 0,Y 509.82,Z 223.474,A -85,B 0,C 180,E1 -5452.658,E2 -5452.658} C_VEL
LIN {X 0,Y 509.867,Z 223.475,A -85,B 0,C 180,E1 -5455.798,E2 -5455.798} C_VEL
LIN {X 0,Y 509.856,Z 223.47,A -85,B 0,C 180,E1 -5458.72,E2 -5458.72} C_VEL
LIN {X 0,Y 509.862,Z 223.471,A -85,B 0,C 180,E1 -5461.154,E2 -5461.154} C_VEL
LIN {X 0,Y 509.878,Z 223.473,A -85,B 0,C 180,E1 -5463.826,E2 -5463.826} C_VEL
LIN {X 0,Y 509.892,Z 223.691,A -85,B 0,C 180,E1 -5466.277,E2 -5466.277} C_VEL
LIN {X 0,Y 511.281,Z 231.843,A -85,B 0,C 180,E1 -5467.788,E2 -5467.788} C_VEL
LIN {X 0,Y 510.852,Z 247.584,A -85,B 0,C 180,E1 -5470.51,E2 -5470.51} C_VEL
LIN {X 0,Y 510.428,Z 263.323,A -85,B 0,C 180,E1 -5473.192,E2 -5473.192} C_VEL
LIN {X 0,Y 510.286,Z 270.668,A -85,B 0,C 180,E1 -5474.397,E2 -5474.397} C_VEL
LIN {X 0,Y 512.228,Z 282.881,A -85,B 0,C 180,E1 -5474.66,E2 -5474.66} C_VEL
LIN {X 0,Y 511.759,Z 379.037,A -85,B 0,C 180,E1 -5476.042,E2 -5476.042} C_VEL
LIN {X 0,Y 511.516,Z 392.077,A -85,B 0,C 180,E1 -5476.39,E2 -5476.39} C_VEL
LIN {X 0,Y 511.171,Z 404.683,A -85,B 0,C 180,E1 -5476.887,E2 -5476.887} C_VEL
LIN {X 0,Y 510.92,Z 416.069,A -85,B 0,C 180,E1 -5477.498,E2 -5477.498} C_VEL
LIN {X 0,Y 510.603,Z 427.512,A -85,B 0,C 180,E1 -5478.285,E2 -5478.285} C_VEL
LIN {X 0,Y 510.218,Z 437.967,A -85,B 0,C 180,E1 -5479.182,E2 -5479.182} C_VEL
LIN {X 0,Y 509.954,Z 446.513,A -85,B 0,C 180,E1 -5480.079,E2 -5480.079} C_VEL
LIN {X 0,Y 509.691,Z 454.395,A -85,B 0,C 180,E1 -5481.075,E2 -5481.075} C_VEL
LIN {X 0,Y 509.506,Z 462.091,A -85,B 0,C 180,E1 -5482.27,E2 -5482.27} C_VEL
LIN {X 0,Y 509.314,Z 469.179,A -85,B 0,C 180,E1 -5483.661,E2 -5483.661} C_VEL
LIN {X 0,Y 509.248,Z 473.894,A -85,B 0,C 180,E1 -5484.852,E2 -5484.852} C_VEL
LIN {X 0,Y 509.247,Z 477.496,A -85,B 0,C 180,E1 -5486.042,E2 -5486.042} C_VEL
LIN {X 0,Y 509.202,Z 479.354,A -85,B 0,C 180,E1 -5486.834,E2 -5486.834} C_VEL
LIN {X 0,Y 509.162,Z 480.747,A -85,B 0,C 180,E1 -5487.626,E2 -5487.626} C_VEL
LIN {X 0,Y 509.074,Z 482.345,A -85,B 0,C 180,E1 -5489.208,E2 -5489.208} C_VEL
LIN {X 0,Y 509.067,Z 482.561,A -85,B 0,C 180,E1 -5489.999,E2 -5489.999} C_VEL
LIN {X 0,Y 509.113,Z 481.741,A -85,B 0,C 180,E1 -5491.581,E2 -5491.581} C_VEL
LIN {X 0,Y 509.162,Z 480.748,A -85,B 0,C 180,E1 -5492.372,E2 -5492.372} C_VEL
LIN {X 0,Y 509.202,Z 479.356,A -85,B 0,C 180,E1 -5493.164,E2 -5493.164} C_VEL
LIN {X 0,Y 509.206,Z 476.427,A -85,B 0,C 180,E1 -5494.352,E2 -5494.352} C_VEL
LIN {X 0,Y 509.311,Z 472.461,A -85,B 0,C 180,E1 -5495.542,E2 -5495.542} C_VEL
LIN {X 0,Y 509.366,Z 466.461,A -85,B 0,C 180,E1 -5496.913,E2 -5496.913} C_VEL
LIN {X 0,Y 509.561,Z 459.69,A -85,B 0,C 180,E1 -5498.126,E2 -5498.126} C_VEL
LIN {X 0,Y 509.77,Z 451.412,A -85,B 0,C 180,E1 -5499.321,E2 -5499.321} C_VEL
LIN {X 0,Y 510.032,Z 442.922,A -85,B 0,C 180,E1 -5500.318,E2 -5500.318} C_VEL
LIN {X 0,Y 510.39,Z 432.429,A -85,B 0,C 180,E1 -5501.315,E2 -5501.315} C_VEL
LIN {X 0,Y 510.721,Z 421.748,A -85,B 0,C 180,E1 -5502.133,E2 -5502.133} C_VEL
LIN {X 0,Y 511.053,Z 410.651,A -85,B 0,C 180,E1 -5502.811,E2 -5502.811} C_VEL
LIN {X 0,Y 511.351,Z 398.927,A -85,B 0,C 180,E1 -5503.359,E2 -5503.359} C_VEL
LIN {X 0,Y 511.581,Z 385.412,A -85,B 0,C 180,E1 -5503.808,E2 -5503.808} C_VEL
LIN {X 0,Y 511.81,Z 371.899,A -85,B 0,C 180,E1 -5504.08,E2 -5504.08} C_VEL
LIN {X 0,Y 512.167,Z 282.488,A -85,B 0,C 180,E1 -5505.347,E2 -5505.347} C_VEL
LIN {X 0,Y 510.287,Z 270.763,A -85,B 0,C 180,E1 -5505.592,E2 -5505.592} C_VEL
LIN {X 0,Y 510.313,Z 266.858,A -85,B 0,C 180,E1 -5506.192,E2 -5506.192} C_VEL
LIN {X 0,Y 510.766,Z 249.828,A -85,B 0,C 180,E1 -5509.073,E2 -5509.073} C_VEL
LIN {X 0,Y 511.28,Z 232.765,A -85,B 0,C 180,E1 -5511.997,E2 -5511.997} C_VEL
LIN {X 0,Y 510.466,Z 226.608,A -85,B 0,C 180,E1 -5513.109,E2 -5513.109} C_VEL
LIN {X 0,Y 509.886,Z 223.568,A -85,B 0,C 180,E1 -5513.721,E2 -5513.721} C_VEL
LIN {X 0,Y 509.879,Z 223.472,A -85,B 0,C 180,E1 -5517.054,E2 -5517.054} C_VEL
LIN {X 0,Y 509.859,Z 223.479,A -85,B 0,C 180,E1 -5519.749,E2 -5519.749} C_VEL
LIN {X 0,Y 509.874,Z 223.467,A -85,B 0,C 180,E1 -5522.772,E2 -5522.772} C_VEL
LIN {X 0,Y 509.823,Z 223.476,A -85,B 0,C 180,E1 -5525.576,E2 -5525.576} C_VEL
LIN {X 0,Y 509.848,Z 223.475,A -85,B 0,C 180,E1 -5528.336,E2 -5528.336} C_VEL
LIN {X 0,Y 509.852,Z 223.47,A -85,B 0,C 180,E1 -5531.424,E2 -5531.424} C_VEL
LIN {X 0,Y 509.838,Z 223.475,A -85,B 0,C 180,E1 -5534.668,E2 -5534.668} C_VEL
LIN {X 0,Y 509.844,Z 223.473,A -85,B 0,C 180,E1 -5538.102,E2 -5538.102} C_VEL
LIN {X 0,Y 509.83,Z 223.479,A -85,B 0,C 180,E1 -5540.644,E2 -5540.644} C_VEL
LIN {X 0,Y 509.806,Z 223.475,A -85,B 0,C 180,E1 -5543.643,E2 -5543.643} C_VEL
LIN {X 0,Y 509.855,Z 223.478,A -85,B 0,C 180,E1 -5546.537,E2 -5546.537} C_VEL
LIN {X 0,Y 509.835,Z 223.473,A -85,B 0,C 180,E1 -5549.331,E2 -5549.331} C_VEL
LIN {X 0,Y 509.84,Z 223.472,A -85,B 0,C 180,E1 -5552.049,E2 -5552.049} C_VEL
LIN {X 0,Y 509.795,Z 223.483,A -85,B 0,C 180,E1 -5554.697,E2 -5554.697} C_VEL
LIN {X 0,Y 509.818,Z 223.476,A -85,B 0,C 180,E1 -5557.456,E2 -5557.456} C_VEL
LIN {X 0,Y 509.9,Z 223.463,A -85,B 0,C 180,E1 -5559.842,E2 -5559.842} C_VEL
LIN {X 0,Y 509.849,Z 223.476,A -85,B 0,C 180,E1 -5563.171,E2 -5563.171} C_VEL
LIN {X 0,Y 509.834,Z 223.475,A -85,B 0,C 180,E1 -5565.631,E2 -5565.631} C_VEL
LIN {X 0,Y 509.896,Z 223.466,A -85,B 0,C 180,E1 -5568.871,E2 -5568.871} C_VEL
LIN {X 0,Y 509.874,Z 223.464,A -85,B 0,C 180,E1 -5572.074,E2 -5572.074} C_VEL
LIN {X 0,Y 509.949,Z 223.458,A -85,B 0,C 180,E1 -5574.461,E2 -5574.461} C_VEL
LIN {X 0,Y 510.022,Z 223.456,A -85,B 0,C 180,E1 -5577.628,E2 -5577.628} C_VEL
LIN {X 0,Y 510.011,Z 223.452,A -85,B 0,C 180,E1 -5579.997,E2 -5579.997} C_VEL
LIN {X 0,Y 510.02,Z 223.449,A -85,B 0,C 180,E1 -5582.366,E2 -5582.366} C_VEL
LIN {X 0,Y 509.917,Z 223.468,A -85,B 0,C 180,E1 -5585.533,E2 -5585.533} C_VEL
LIN {X 0,Y 509.881,Z 223.466,A -85,B 0,C 180,E1 -5588.717,E2 -5588.717} C_VEL
LIN {X 0,Y 509.883,Z 223.474,A -85,B 0,C 180,E1 -5591.929,E2 -5591.929} C_VEL
LIN {X 0,Y 509.872,Z 223.469,A -85,B 0,C 180,E1 -5595.239,E2 -5595.239} C_VEL
LIN {X 0,Y 509.832,Z 223.476,A -85,B 0,C 180,E1 -5598.481,E2 -5598.481} C_VEL
LIN {X 0,Y 509.824,Z 223.474,A -85,B 0,C 180,E1 -5600.999,E2 -5600.999} C_VEL
LIN {X 0,Y 509.795,Z 223.479,A -85,B 0,C 180,E1 -5603.561,E2 -5603.561} C_VEL
LIN {X 0,Y 509.881,Z 223.475,A -85,B 0,C 180,E1 -5606.375,E2 -5606.375} C_VEL
LIN {X 0,Y 509.846,Z 223.471,A -85,B 0,C 180,E1 -5608.841,E2 -5608.841} C_VEL
LIN {X 0,Y 509.79,Z 223.479,A -85,B 0,C 180,E1 -5611.587,E2 -5611.587} C_VEL
LIN {X 0,Y 509.821,Z 223.483,A -85,B 0,C 180,E1 -5614.411,E2 -5614.411} C_VEL
LIN {X 0,Y 509.786,Z 223.48,A -85,B 0,C 180,E1 -5617.338,E2 -5617.338} C_VEL
LIN {X 0,Y 509.827,Z 223.48,A -85,B 0,C 180,E1 -5620.377,E2 -5620.377} C_VEL
LIN {X 0,Y 509.803,Z 223.482,A -85,B 0,C 180,E1 -5623.062,E2 -5623.062} C_VEL
LIN {X 0,Y 509.793,Z 223.482,A -85,B 0,C 180,E1 -5625.79,E2 -5625.79} C_VEL
LIN {X 0,Y 509.851,Z 223.581,A -85,B 0,C 180,E1 -5627.344,E2 -5627.344} C_VEL
LIN {X 0,Y 510.73,Z 228.69,A -85,B 0,C 180,E1 -5628.351,E2 -5628.351} C_VEL
LIN {X 0,Y 510.516,Z 243.26,A -85,B 0,C 180,E1 -5630.966,E2 -5630.966} C_VEL
LIN {X 0,Y 510.295,Z 253.149,A -85,B 0,C 180,E1 -5632.731,E2 -5632.731} C_VEL
LIN {X 0,Y 510.003,Z 255.701,A -85,B 0,C 180,E1 -5633.047,E2 -5633.047} C_VEL
LIN {X 0,Y 509.36,Z 258.924,A -85,B 0,C 180,E1 -5633.273,E2 -5633.273} C_VEL
LIN {X 0,Y 508.08,Z 264.436,A -85,B 0,C 180,E1 -5633.478,E2 -5633.478} C_VEL
LIN {X 0,Y 505.625,Z 276.818,A -85,B 0,C 180,E1 -5633.602,E2 -5633.602} C_VEL
LIN {X 0,Y 505.322,Z 283.178,A -85,B 0,C 180,E1 -5633.688,E2 -5633.688} C_VEL
LIN {X 0,Y 504.888,Z 364.911,A -85,B 0,C 180,E1 -5634.882,E2 -5634.882} C_VEL
LIN {X 0,Y 504.626,Z 378.431,A -85,B 0,C 180,E1 -5635.247,E2 -5635.247} C_VEL
LIN {X 0,Y 504.368,Z 391.281,A -85,B 0,C 180,E1 -5635.766,E2 -5635.766} C_VEL
LIN {X 0,Y 504.013,Z 402.992,A -85,B 0,C 180,E1 -5636.411,E2 -5636.411} C_VEL
LIN {X 0,Y 503.583,Z 414.995,A -85,B 0,C 180,E1 -5637.264,E2 -5637.264} C_VEL
LIN {X 0,Y 503.25,Z 425.667,A -85,B 0,C 180,E1 -5638.224,E2 -5638.224} C_VEL
LIN {X 0,Y 502.897,Z 435.52,A -85,B 0,C 180,E1 -5639.332,E2 -5639.332} C_VEL
LIN {X 0,Y 502.593,Z 444.195,A -85,B 0,C 180,E1 -5640.539,E2 -5640.539} C_VEL
LIN {X 0,Y 502.453,Z 451.268,A -85,B 0,C 180,E1 -5641.777,E2 -5641.777} C_VEL
LIN {X 0,Y 502.287,Z 456.667,A -85,B 0,C 180,E1 -5642.953,E2 -5642.953} C_VEL
LIN {X 0,Y 502.15,Z 461.431,A -85,B 0,C 180,E1 -5644.288,E2 -5644.288} C_VEL
LIN {X 0,Y 502.084,Z 464.574,A -85,B 0,C 180,E1 -5645.472,E2 -5645.472} C_VEL
LIN {X 0,Y 501.966,Z 467.152,A -85,B 0,C 180,E1 -5646.921,E2 -5646.921} C_VEL
LIN {X 0,Y 501.97,Z 468.073,A -85,B 0,C 180,E1 -5647.79,E2 -5647.79} C_VEL
LIN {X 0,Y 501.936,Z 468.486,A -85,B 0,C 180,E1 -5648.653,E2 -5648.653} C_VEL
LIN {X 0,Y 501.996,Z 468.421,A -85,B 0,C 180,E1 -5649.704,E2 -5649.704} C_VEL
LIN {X 0,Y 501.996,Z 467.076,A -85,B 0,C 180,E1 -5651.217,E2 -5651.217} C_VEL
LIN {X 0,Y 502.022,Z 465.556,A -85,B 0,C 180,E1 -5652.151,E2 -5652.151} C_VEL
LIN {X 0,Y 502.11,Z 462.804,A -85,B 0,C 180,E1 -5653.327,E2 -5653.327} C_VEL
LIN {X 0,Y 502.198,Z 458.81,A -85,B 0,C 180,E1 -5654.581,E2 -5654.581} C_VEL
LIN {X 0,Y 502.339,Z 453.634,A -85,B 0,C 180,E1 -5655.829,E2 -5655.829} C_VEL
LIN {X 0,Y 502.493,Z 447.113,A -85,B 0,C 180,E1 -5657.07,E2 -5657.07} C_VEL
LIN {X 0,Y 502.776,Z 439.543,A -85,B 0,C 180,E1 -5658.226,E2 -5658.226} C_VEL
LIN {X 0,Y 503.067,Z 430.634,A -85,B 0,C 180,E1 -5659.334,E2 -5659.334} C_VEL
LIN {X 0,Y 503.436,Z 420.483,A -85,B 0,C 180,E1 -5660.358,E2 -5660.358} C_VEL
LIN {X 0,Y 503.778,Z 410.413,A -85,B 0,C 180,E1 -5661.174,E2 -5661.174} C_VEL
LIN {X 0,Y 504.124,Z 399.389,A -85,B 0,C 180,E1 -5661.891,E2 -5661.891} C_VEL
LIN {X 0,Y 504.478,Z 387.359,A -85,B 0,C 180,E1 -5662.497,E2 -5662.497} C_VEL
LIN {X 0,Y 504.7,Z 374.982,A -85,B 0,C 180,E1 -5662.953,E2 -5662.953} C_VEL
LIN {X 0,Y 504.879,Z 362.106,A -85,B 0,C 180,E1 -5663.256,E2 -5663.256} C_VEL
LIN {X 0,Y 505.275,Z 269.04,A -85,B 0,C 180,E1 -5664.602,E2 -5664.602} C_VEL
LIN {X 0,Y 503.294,Z 257.906,A -85,B 0,C 180,E1 -5664.844,E2 -5664.844} C_VEL
LIN {X 0,Y 503.26,Z 256.694,A -85,B 0,C 180,E1 -5664.994,E2 -5664.994} C_VEL
LIN {X 0,Y 503.731,Z 240.6,A -85,B 0,C 180,E1 -5668.002,E2 -5668.002} C_VEL
LIN {X 0,Y 504.001,Z 231.11,A -85,B 0,C 180,E1 -5669.802,E2 -5669.802} C_VEL
LIN {X 0,Y 502.958,Z 224.677,A -85,B 0,C 180,E1 -5671.102,E2 -5671.102} C_VEL
LIN {X 0,Y 502.874,Z 224.348,A -85,B 0,C 180,E1 -5671.403,E2 -5671.403} C_VEL
LIN {X 0,Y 502.862,Z 224.349,A -85,B 0,C 180,E1 -5673.206,E2 -5673.206} C_VEL
LIN {X 0,Y 502.864,Z 224.343,A -85,B 0,C 180,E1 -5676.421,E2 -5676.421} C_VEL
LIN {X 0,Y 502.83,Z 224.345,A -85,B 0,C 180,E1 -5678.845,E2 -5678.845} C_VEL
LIN {X 0,Y 502.851,Z 224.344,A -85,B 0,C 180,E1 -5682.103,E2 -5682.103} C_VEL
LIN {X 0,Y 502.807,Z 224.352,A -85,B 0,C 180,E1 -5685.402,E2 -5685.402} C_VEL
LIN {X 0,Y 502.806,Z 224.352,A -85,B 0,C 180,E1 -5688.125,E2 -5688.125} C_VEL
LIN {X 0,Y 502.79,Z 224.351,A -85,B 0,C 180,E1 -5690.539,E2 -5690.539} C_VEL
LIN {X 0,Y 502.749,Z 224.354,A -85,B 0,C 180,E1 -5693.044,E2 -5693.044} C_VEL
LIN {X 0,Y 502.753,Z 224.358,A -85,B 0,C 180,E1 -5695.681,E2 -5695.681} C_VEL
LIN {X 0,Y 502.76,Z 224.359,A -85,B 0,C 180,E1 -5698.379,E2 -5698.379} C_VEL
LIN {X 0,Y 502.762,Z 224.353,A -85,B 0,C 180,E1 -5701.147,E2 -5701.147} C_VEL
LIN {X 0,Y 502.753,Z 224.358,A -85,B 0,C 180,E1 -5703.999,E2 -5703.999} C_VEL
LIN {X 0,Y 502.72,Z 224.359,A -85,B 0,C 180,E1 -5707.177,E2 -5707.177} C_VEL
LIN {X 0,Y 502.742,Z 224.358,A -85,B 0,C 180,E1 -5710.021,E2 -5710.021} C_VEL
LIN {X 0,Y 502.724,Z 224.359,A -85,B 0,C 180,E1 -5713.238,E2 -5713.238} C_VEL
LIN {X 0,Y 502.755,Z 224.354,A -85,B 0,C 180,E1 -5715.664,E2 -5715.664} C_VEL
LIN {X 0,Y 502.773,Z 224.351,A -85,B 0,C 180,E1 -5717.865,E2 -5717.865} C_VEL
LIN {X 0,Y 502.773,Z 224.359,A -85,B 0,C 180,E1 -5721.027,E2 -5721.027} C_VEL
LIN {X 0,Y 502.757,Z 224.354,A -85,B 0,C 180,E1 -5724.173,E2 -5724.173} C_VEL
LIN {X 0,Y 502.788,Z 224.358,A -85,B 0,C 180,E1 -5727.003,E2 -5727.003} C_VEL
LIN {X 0,Y 502.796,Z 224.349,A -85,B 0,C 180,E1 -5730.07,E2 -5730.07} C_VEL
LIN {X 0,Y 502.771,Z 224.359,A -85,B 0,C 180,E1 -5733.433,E2 -5733.433} C_VEL
LIN {X 0,Y 502.757,Z 224.354,A -85,B 0,C 180,E1 -5736.089,E2 -5736.089} C_VEL
LIN {X 0,Y 502.777,Z 224.351,A -85,B 0,C 180,E1 -5738.693,E2 -5738.693} C_VEL
LIN {X 0,Y 502.806,Z 224.352,A -85,B 0,C 180,E1 -5741.251,E2 -5741.251} C_VEL
LIN {X 0,Y 502.835,Z 224.344,A -85,B 0,C 180,E1 -5744.668,E2 -5744.668} C_VEL
LIN {X 0,Y 502.869,Z 224.345,A -85,B 0,C 180,E1 -5748.047,E2 -5748.047} C_VEL
LIN {X 0,Y 502.848,Z 224.343,A -85,B 0,C 180,E1 -5751.16,E2 -5751.16} C_VEL
LIN {X 0,Y 502.869,Z 224.344,A -85,B 0,C 180,E1 -5753.584,E2 -5753.584} C_VEL
LIN {X 0,Y 502.838,Z 224.344,A -85,B 0,C 180,E1 -5756.798,E2 -5756.798} C_VEL
LIN {X 0,Y 502.901,Z 224.34,A -85,B 0,C 180,E1 -5758.402,E2 -5758.402} C_VEL
LIN {X 0,Y 502.975,Z 224.328,A -85,B 0,C 180,E1 -5760.804,E2 -5760.804} C_VEL
LIN {X 0,Y 503.013,Z 224.329,A -85,B 0,C 180,E1 -5762.405,E2 -5762.405} C_VEL
LIN {X 0,Y 502.903,Z 224.336,A -85,B 0,C 180,E1 -5765.617,E2 -5765.617} C_VEL
LIN {X 0,Y 502.855,Z 224.345,A -85,B 0,C 180,E1 -5768.037,E2 -5768.037} C_VEL
LIN {X 0,Y 502.883,Z 224.338,A -85,B 0,C 180,E1 -5771.286,E2 -5771.286} C_VEL
LIN {X 0,Y 502.839,Z 224.352,A -85,B 0,C 180,E1 -5774.574,E2 -5774.574} C_VEL
LIN {X 0,Y 502.821,Z 224.35,A -85,B 0,C 180,E1 -5777.071,E2 -5777.071} C_VEL
LIN {X 0,Y 502.824,Z 224.345,A -85,B 0,C 180,E1 -5779.602,E2 -5779.602} C_VEL
LIN {X 0,Y 502.815,Z 224.353,A -85,B 0,C 180,E1 -5782.703,E2 -5782.703} C_VEL
LIN {X 0,Y 502.791,Z 224.35,A -85,B 0,C 180,E1 -5785.681,E2 -5785.681} C_VEL
LIN {X 0,Y 502.786,Z 224.351,A -85,B 0,C 180,E1 -5788.378,E2 -5788.378} C_VEL
LIN {X 0,Y 502.801,Z 224.358,A -85,B 0,C 180,E1 -5791.145,E2 -5791.145} C_VEL
LIN {X 0,Y 502.799,Z 224.349,A -85,B 0,C 180,E1 -5793.996,E2 -5793.996} C_VEL
LIN {X 0,Y 502.776,Z 224.358,A -85,B 0,C 180,E1 -5797.176,E2 -5797.176} C_VEL
LIN {X 0,Y 502.786,Z 224.352,A -85,B 0,C 180,E1 -5800.018,E2 -5800.018} C_VEL
LIN {X 0,Y 502.761,Z 224.357,A -85,B 0,C 180,E1 -5803.235,E2 -5803.235} C_VEL
LIN {X 0,Y 502.793,Z 224.359,A -85,B 0,C 180,E1 -5805.66,E2 -5805.66} C_VEL
LIN {X 0,Y 502.778,Z 224.351,A -85,B 0,C 180,E1 -5809.013,E2 -5809.013} C_VEL
LIN {X 0,Y 502.802,Z 224.354,A -85,B 0,C 180,E1 -5812.046,E2 -5812.046} C_VEL
LIN {X 0,Y 502.809,Z 224.347,A -85,B 0,C 180,E1 -5815.034,E2 -5815.034} C_VEL
LIN {X 0,Y 502.795,Z 224.356,A -85,B 0,C 180,E1 -5817.915,E2 -5817.915} C_VEL
LIN {X 0,Y 502.825,Z 224.35,A -85,B 0,C 180,E1 -5820.711,E2 -5820.711} C_VEL
LIN {X 0,Y 502.856,Z 224.345,A -85,B 0,C 180,E1 -5823.443,E2 -5823.443} C_VEL
LIN {X 0,Y 502.85,Z 224.512,A -85,B 0,C 180,E1 -5826.088,E2 -5826.088} C_VEL
LIN {X 0,Y 504.326,Z 232.947,A -85,B 0,C 180,E1 -5827.681,E2 -5827.681} C_VEL
LIN {X 0,Y 503.899,Z 247.477,A -85,B 0,C 180,E1 -5830.23,E2 -5830.23} C_VEL
LIN {X 0,Y 503.505,Z 262.004,A -85,B 0,C 180,E1 -5832.745,E2 -5832.745} C_VEL
LIN {X 0,Y 503.295,Z 270.508,A -85,B 0,C 180,E1 -5834.173,E2 -5834.173} C_VEL
LIN {X 0,Y 504.319,Z 276.969,A -85,B 0,C 180,E1 -5834.332,E2 -5834.332} C_VEL
LIN {X 0,Y 505.406,Z 285.185,A -85,B 0,C 180,E1 -5834.484,E2 -5834.484} C_VEL
LIN {X 0,Y 504.868,Z 378.875,A -85,B 0,C 180,E1 -5835.848,E2 -5835.848} C_VEL
LIN {X 0,Y 504.598,Z 391.936,A -85,B 0,C 180,E1 -5836.2,E2 -5836.2} C_VEL
LIN {X 0,Y 504.239,Z 404.553,A -85,B 0,C 180,E1 -5836.703,E2 -5836.703} C_VEL
LIN {X 0,Y 503.949,Z 416.686,A -85,B 0,C 180,E1 -5837.37,E2 -5837.37} C_VEL
LIN {X 0,Y 503.598,Z 428.69,A -85,B 0,C 180,E1 -5838.222,E2 -5838.222} C_VEL
LIN {X 0,Y 503.184,Z 438.906,A -85,B 0,C 180,E1 -5839.13,E2 -5839.13} C_VEL
LIN {X 0,Y 502.876,Z 448.088,A -85,B 0,C 180,E1 -5840.141,E2 -5840.141} C_VEL
LIN {X 0,Y 502.601,Z 457.028,A -85,B 0,C 180,E1 -5841.353,E2 -5841.353} C_VEL
LIN {X 0,Y 502.361,Z 464.223,A -85,B 0,C 180,E1 -5842.563,E2 -5842.563} C_VEL
LIN {X 0,Y 502.242,Z 469.077,A -85,B 0,C 180,E1 -5843.571,E2 -5843.571} C_VEL
LIN {X 0,Y 502.182,Z 473.794,A -85,B 0,C 180,E1 -5844.78,E2 -5844.78} C_VEL
LIN {X 0,Y 502.141,Z 477.397,A -85,B 0,C 180,E1 -5845.986,E2 -5845.986} C_VEL
LIN {X 0,Y 502.122,Z 479.255,A -85,B 0,C 180,E1 -5846.789,E2 -5846.789} C_VEL
LIN {X 0,Y 502.067,Z 480.648,A -85,B 0,C 180,E1 -5847.592,E2 -5847.592} C_VEL
LIN {X 0,Y 502.037,Z 481.641,A -85,B 0,C 180,E1 -5848.394,E2 -5848.394} C_VEL
LIN {X 0,Y 501.982,Z 482.463,A -85,B 0,C 180,E1 -5849.999,E2 -5849.999} C_VEL
LIN {X 0,Y 502.037,Z 481.642,A -85,B 0,C 180,E1 -5851.603,E2 -5851.603} C_VEL
LIN {X 0,Y 502.067,Z 480.649,A -85,B 0,C 180,E1 -5852.406,E2 -5852.406} C_VEL
LIN {X 0,Y 502.122,Z 479.256,A -85,B 0,C 180,E1 -5853.208,E2 -5853.208} C_VEL
LIN {X 0,Y 502.104,Z 476.325,A -85,B 0,C 180,E1 -5854.414,E2 -5854.414} C_VEL
LIN {X 0,Y 502.229,Z 472.358,A -85,B 0,C 180,E1 -5855.62,E2 -5855.62} C_VEL
LIN {X 0,Y 502.291,Z 466.354,A -85,B 0,C 180,E1 -5857.011,E2 -5857.011} C_VEL
LIN {X 0,Y 502.492,Z 459.581,A -85,B 0,C 180,E1 -5858.241,E2 -5858.241} C_VEL
LIN {X 0,Y 502.742,Z 451.301,A -85,B 0,C 180,E1 -5859.453,E2 -5859.453} C_VEL
LIN {X 0,Y 503.018,Z 442.807,A -85,B 0,C 180,E1 -5860.463,E2 -5860.463} C_VEL
LIN {X 0,Y 503.431,Z 432.309,A -85,B 0,C 180,E1 -5861.473,E2 -5861.473} C_VEL
LIN {X 0,Y 503.747,Z 421.624,A -85,B 0,C 180,E1 -5862.304,E2 -5862.304} C_VEL
LIN {X 0,Y 504.11,Z 410.532,A -85,B 0,C 180,E1 -5862.99,E2 -5862.99} C_VEL
LIN {X 0,Y 504.426,Z 398.818,A -85,B 0,C 180,E1 -5863.546,E2 -5863.546} C_VEL
LIN {X 0,Y 504.693,Z 385.322,A -85,B 0,C 180,E1 -5864,E2 -5864} C_VEL
LIN {X 0,Y 504.947,Z 371.849,A -85,B 0,C 180,E1 -5864.276,E2 -5864.276} C_VEL
LIN {X 0,Y 505.312,Z 282.993,A -85,B 0,C 180,E1 -5865.555,E2 -5865.555} C_VEL
LIN {X 0,Y 503.282,Z 270.592,A -85,B 0,C 180,E1 -5865.823,E2 -5865.823} C_VEL
LIN {X 0,Y 503.401,Z 264.345,A -85,B 0,C 180,E1 -5866.838,E2 -5866.838} C_VEL
LIN {X 0,Y 503.836,Z 248.52,A -85,B 0,C 180,E1 -5869.557,E2 -5869.557} C_VEL
LIN {X 0,Y 504.35,Z 233.893,A -85,B 0,C 180,E1 -5872.099,E2 -5872.099} C_VEL
LIN {X 0,Y 503.264,Z 226.593,A -85,B 0,C 180,E1 -5873.451,E2 -5873.451} C_VEL
LIN {X 0,Y 502.853,Z 224.441,A -85,B 0,C 180,E1 -5873.909,E2 -5873.909} C_VEL
LIN {X 0,Y 502.84,Z 224.348,A -85,B 0,C 180,E1 -5876.566,E2 -5876.566} C_VEL
LIN {X 0,Y 502.824,Z 224.349,A -85,B 0,C 180,E1 -5879.286,E2 -5879.286} C_VEL
LIN {X 0,Y 502.784,Z 224.356,A -85,B 0,C 180,E1 -5882.083,E2 -5882.083} C_VEL
LIN {X 0,Y 502.798,Z 224.348,A -85,B 0,C 180,E1 -5884.964,E2 -5884.964} C_VEL
LIN {X 0,Y 502.792,Z 224.353,A -85,B 0,C 180,E1 -5888.483,E2 -5888.483} C_VEL
LIN {X 0,Y 502.799,Z 224.348,A -85,B 0,C 180,E1 -5891.066,E2 -5891.066} C_VEL
LIN {X 0,Y 502.778,Z 224.359,A -85,B 0,C 180,E1 -5894.338,E2 -5894.338} C_VEL
LIN {X 0,Y 502.756,Z 224.353,A -85,B 0,C 180,E1 -5896.765,E2 -5896.765} C_VEL
LIN {X 0,Y 502.773,Z 224.354,A -85,B 0,C 180,E1 -5899.009,E2 -5899.009} C_VEL
LIN {X 0,Y 502.787,Z 224.354,A -85,B 0,C 180,E1 -5902.043,E2 -5902.043} C_VEL
LIN {X 0,Y 502.794,Z 224.353,A -85,B 0,C 180,E1 -5905.032,E2 -5905.032} C_VEL
LIN {X 0,Y 502.778,Z 224.351,A -85,B 0,C 180,E1 -5907.913,E2 -5907.913} C_VEL
LIN {X 0,Y 502.807,Z 224.354,A -85,B 0,C 180,E1 -5910.709,E2 -5910.709} C_VEL
LIN {X 0,Y 502.769,Z 224.353,A -85,B 0,C 180,E1 -5913.457,E2 -5913.457} C_VEL
LIN {X 0,Y 502.759,Z 224.354,A -85,B 0,C 180,E1 -5916.082,E2 -5916.082} C_VEL
LIN {X 0,Y 502.772,Z 224.357,A -85,B 0,C 180,E1 -5918.686,E2 -5918.686} C_VEL
LIN {X 0,Y 502.813,Z 224.352,A -85,B 0,C 180,E1 -5921.245,E2 -5921.245} C_VEL
LIN {X 0,Y 502.829,Z 224.347,A -85,B 0,C 180,E1 -5924.661,E2 -5924.661} C_VEL
LIN {X 0,Y 502.867,Z 224.338,A -85,B 0,C 180,E1 -5928.036,E2 -5928.036} C_VEL
LIN {X 0,Y 502.825,Z 224.354,A -85,B 0,C 180,E1 -5931.153,E2 -5931.153} C_VEL
LIN {X 0,Y 502.875,Z 224.345,A -85,B 0,C 180,E1 -5933.578,E2 -5933.578} C_VEL
LIN {X 0,Y 502.817,Z 224.345,A -85,B 0,C 180,E1 -5936.792,E2 -5936.792} C_VEL
LIN {X 0,Y 502.872,Z 224.34,A -85,B 0,C 180,E1 -5938.395,E2 -5938.395} C_VEL
LIN {X 0,Y 502.98,Z 224.328,A -85,B 0,C 180,E1 -5939.997,E2 -5939.997} C_VEL
LIN {X 0,Y 502.989,Z 224.325,A -85,B 0,C 180,E1 -5942.399,E2 -5942.399} C_VEL
LIN {X 0,Y 502.873,Z 224.345,A -85,B 0,C 180,E1 -5945.611,E2 -5945.611} C_VEL
LIN {X 0,Y 502.852,Z 224.346,A -85,B 0,C 180,E1 -5948.031,E2 -5948.031} C_VEL
LIN {X 0,Y 502.855,Z 224.344,A -85,B 0,C 180,E1 -5951.28,E2 -5951.28} C_VEL
LIN {X 0,Y 502.808,Z 224.35,A -85,B 0,C 180,E1 -5954.568,E2 -5954.568} C_VEL
LIN {X 0,Y 502.792,Z 224.356,A -85,B 0,C 180,E1 -5957.906,E2 -5957.906} C_VEL
LIN {X 0,Y 502.804,Z 224.352,A -85,B 0,C 180,E1 -5960.533,E2 -5960.533} C_VEL
LIN {X 0,Y 502.761,Z 224.354,A -85,B 0,C 180,E1 -5963.038,E2 -5963.038} C_VEL
LIN {X 0,Y 502.791,Z 224.351,A -85,B 0,C 180,E1 -5965.674,E2 -5965.674} C_VEL
LIN {X 0,Y 502.81,Z 224.35,A -85,B 0,C 180,E1 -5968.37,E2 -5968.37} C_VEL
LIN {X 0,Y 502.762,Z 224.354,A -85,B 0,C 180,E1 -5971.496,E2 -5971.496} C_VEL
LIN {X 0,Y 502.774,Z 224.361,A -85,B 0,C 180,E1 -5974.442,E2 -5974.442} C_VEL
LIN {X 0,Y 502.748,Z 224.358,A -85,B 0,C 180,E1 -5977.176,E2 -5977.176} C_VEL
LIN {X 0,Y 502.791,Z 224.353,A -85,B 0,C 180,E1 -5980.009,E2 -5980.009} C_VEL
LIN {X 0,Y 502.79,Z 224.355,A -85,B 0,C 180,E1 -5982.2,E2 -5982.2} C_VEL
LIN {X 0,Y 502.762,Z 224.359,A -85,B 0,C 180,E1 -5985.466,E2 -5985.466} C_VEL
LIN {X 0,Y 502.809,Z 224.428,A -85,B 0,C 180,E1 -5987.172,E2 -5987.172} C_VEL
LIN {X 0,Y 503.79,Z 230.185,A -85,B 0,C 180,E1 -5988.323,E2 -5988.323} C_VEL
LIN {X 0,Y 503.551,Z 244.003,A -85,B 0,C 180,E1 -5990.838,E2 -5990.838} C_VEL
LIN {X 0,Y 503.285,Z 257.34,A -85,B 0,C 180,E1 -5993.204,E2 -5993.204} C_VEL
LIN {X 0,Y 503.979,Z 261.433,A -85,B 0,C 180,E1 -5993.326,E2 -5993.326} C_VEL
LIN {X 0,Y 505.442,Z 270.825,A -85,B 0,C 180,E1 -5993.512,E2 -5993.512} C_VEL
LIN {X 0,Y 505.322,Z 283.178,A -85,B 0,C 180,E1 -5993.688,E2 -5993.688} C_VEL
LIN {X 0,Y 504.658,Z 289.021,A -85,B 0,C 180,E1 -5993.752,E2 -5993.752} C_VEL
LIN {X 0,Y 499.032,Z 308.026,A -85,B 0,C 180,E1 -5993.85,E2 -5993.85} C_VEL
LIN {X 0,Y 498.324,Z 313.871,A -85,B 0,C 180,E1 -5993.914,E2 -5993.914} C_VEL
LIN {X 0,Y 498.007,Z 364.88,A -85,B 0,C 180,E1 -5994.676,E2 -5994.676} C_VEL
LIN {X 0,Y 497.746,Z 378.481,A -85,B 0,C 180,E1 -5995.047,E2 -5995.047} C_VEL
LIN {X 0,Y 497.49,Z 390.679,A -85,B 0,C 180,E1 -5995.543,E2 -5995.543} C_VEL
LIN {X 0,Y 497.129,Z 402.295,A -85,B 0,C 180,E1 -5996.177,E2 -5996.177} C_VEL
LIN {X 0,Y 496.7,Z 413.843,A -85,B 0,C 180,E1 -5996.994,E2 -5996.994} C_VEL
LIN {X 0,Y 496.32,Z 424.699,A -85,B 0,C 180,E1 -5997.959,E2 -5997.959} C_VEL
LIN {X 0,Y 495.983,Z 432.933,A -85,B 0,C 180,E1 -5998.857,E2 -5998.857} C_VEL
LIN {X 0,Y 495.683,Z 441.861,A -85,B 0,C 180,E1 -6000.048,E2 -6000.048} C_VEL
LIN {X 0,Y 495.451,Z 448.691,A -85,B 0,C 180,E1 -6001.167,E2 -6001.167} C_VEL
LIN {X 0,Y 495.23,Z 455.393,A -85,B 0,C 180,E1 -6002.536,E2 -6002.536} C_VEL
LIN {X 0,Y 495.126,Z 460.535,A -85,B 0,C 180,E1 -6003.896,E2 -6003.896} C_VEL
LIN {X 0,Y 494.992,Z 464.435,A -85,B 0,C 180,E1 -6005.312,E2 -6005.312} C_VEL
LIN {X 0,Y 494.895,Z 466.812,A -85,B 0,C 180,E1 -6006.572,E2 -6006.572} C_VEL
LIN {X 0,Y 494.881,Z 467.877,A -85,B 0,C 180,E1 -6007.455,E2 -6007.455} C_VEL
LIN {X 0,Y 494.839,Z 468.501,A -85,B 0,C 180,E1 -6008.331,E2 -6008.331} C_VEL
LIN {X 0,Y 494.889,Z 468.554,A -85,B 0,C 180,E1 -6009.584,E2 -6009.584} C_VEL
LIN {X 0,Y 494.917,Z 467.572,A -85,B 0,C 180,E1 -6010.938,E2 -6010.938} C_VEL
LIN {X 0,Y 494.916,Z 465.909,A -85,B 0,C 180,E1 -6012.051,E2 -6012.051} C_VEL
LIN {X 0,Y 495.04,Z 462.591,A -85,B 0,C 180,E1 -6013.506,E2 -6013.506} C_VEL
LIN {X 0,Y 495.155,Z 458.37,A -85,B 0,C 180,E1 -6014.811,E2 -6014.811} C_VEL
LIN {X 0,Y 495.306,Z 452.155,A -85,B 0,C 180,E1 -6016.252,E2 -6016.252} C_VEL
LIN {X 0,Y 495.52,Z 445.244,A -85,B 0,C 180,E1 -6017.51,E2 -6017.51} C_VEL
LIN {X 0,Y 495.754,Z 438.2,A -85,B 0,C 180,E1 -6018.554,E2 -6018.554} C_VEL
LIN {X 0,Y 496.095,Z 429.705,A -85,B 0,C 180,E1 -6019.595,E2 -6019.595} C_VEL
LIN {X 0,Y 496.476,Z 419.235,A -85,B 0,C 180,E1 -6020.632,E2 -6020.632} C_VEL
LIN {X 0,Y 496.95,Z 407.779,A -85,B 0,C 180,E1 -6021.536,E2 -6021.536} C_VEL
LIN {X 0,Y 497.269,Z 397.146,A -85,B 0,C 180,E1 -6022.203,E2 -6022.203} C_VEL
LIN {X 0,Y 497.607,Z 384.623,A -85,B 0,C 180,E1 -6022.801,E2 -6022.801} C_VEL
LIN {X 0,Y 497.861,Z 371.7,A -85,B 0,C 180,E1 -6023.237,E2 -6023.237} C_VEL
LIN {X 0,Y 498.029,Z 359.635,A -85,B 0,C 180,E1 -6023.494,E2 -6023.494} C_VEL
LIN {X 0,Y 498.407,Z 269.721,A -85,B 0,C 180,E1 -6024.806,E2 -6024.806} C_VEL
LIN {X 0,Y 496.302,Z 257.778,A -85,B 0,C 180,E1 -6025.076,E2 -6025.076} C_VEL
LIN {X 0,Y 496.571,Z 248.593,A -85,B 0,C 180,E1 -6026.756,E2 -6026.756} C_VEL
LIN {X 0,Y 497.059,Z 232.696,A -85,B 0,C 180,E1 -6029.799,E2 -6029.799} C_VEL
LIN {X 0,Y 495.871,Z 225.367,A -85,B 0,C 180,E1 -6031.321,E2 -6031.321} C_VEL
LIN {X 0,Y 495.807,Z 225.228,A -85,B 0,C 180,E1 -6033.252,E2 -6033.252} C_VEL
LIN {X 0,Y 495.818,Z 225.221,A -85,B 0,C 180,E1 -6036.512,E2 -6036.512} C_VEL
LIN {X 0,Y 495.799,Z 225.222,A -85,B 0,C 180,E1 -6038.972,E2 -6038.972} C_VEL
LIN {X 0,Y 495.809,Z 225.22,A -85,B 0,C 180,E1 -6042.277,E2 -6042.277} C_VEL
LIN {X 0,Y 495.766,Z 225.232,A -85,B 0,C 180,E1 -6045.626,E2 -6045.626} C_VEL
LIN {X 0,Y 495.767,Z 225.227,A -85,B 0,C 180,E1 -6048.25,E2 -6048.25} C_VEL
LIN {X 0,Y 495.736,Z 225.228,A -85,B 0,C 180,E1 -6050.759,E2 -6050.759} C_VEL
LIN {X 0,Y 495.704,Z 225.234,A -85,B 0,C 180,E1 -6053.391,E2 -6053.391} C_VEL
LIN {X 0,Y 495.723,Z 225.231,A -85,B 0,C 180,E1 -6056.737,E2 -6056.737} C_VEL
LIN {X 0,Y 495.729,Z 225.232,A -85,B 0,C 180,E1 -6059.75,E2 -6059.75} C_VEL
LIN {X 0,Y 495.719,Z 225.235,A -85,B 0,C 180,E1 -6062.599,E2 -6062.599} C_VEL
LIN {X 0,Y 495.706,Z 225.232,A -85,B 0,C 180,E1 -6065.542,E2 -6065.542} C_VEL
LIN {X 0,Y 495.711,Z 225.236,A -85,B 0,C 180,E1 -6068.768,E2 -6068.768} C_VEL
LIN {X 0,Y 495.698,Z 225.233,A -85,B 0,C 180,E1 -6071.788,E2 -6071.788} C_VEL
LIN {X 0,Y 495.713,Z 225.234,A -85,B 0,C 180,E1 -6075.145,E2 -6075.145} C_VEL
LIN {X 0,Y 495.721,Z 225.232,A -85,B 0,C 180,E1 -6078.222,E2 -6078.222} C_VEL
LIN {X 0,Y 495.726,Z 225.232,A -85,B 0,C 180,E1 -6081.412,E2 -6081.412} C_VEL
LIN {X 0,Y 495.73,Z 225.231,A -85,B 0,C 180,E1 -6084.466,E2 -6084.466} C_VEL
LIN {X 0,Y 495.736,Z 225.233,A -85,B 0,C 180,E1 -6087.408,E2 -6087.408} C_VEL
LIN {X 0,Y 495.744,Z 225.227,A -85,B 0,C 180,E1 -6090.257,E2 -6090.257} C_VEL
LIN {X 0,Y 495.727,Z 225.239,A -85,B 0,C 180,E1 -6093.275,E2 -6093.275} C_VEL
LIN {X 0,Y 495.73,Z 225.229,A -85,B 0,C 180,E1 -6096.616,E2 -6096.616} C_VEL
LIN {X 0,Y 495.773,Z 225.231,A -85,B 0,C 180,E1 -6099.328,E2 -6099.328} C_VEL
LIN {X 0,Y 495.775,Z 225.229,A -85,B 0,C 180,E1 -6101.832,E2 -6101.832} C_VEL
LIN {X 0,Y 495.778,Z 225.226,A -85,B 0,C 180,E1 -6105.221,E2 -6105.221} C_VEL
LIN {X 0,Y 495.821,Z 225.218,A -85,B 0,C 180,E1 -6108.558,E2 -6108.558} C_VEL
LIN {X 0,Y 495.815,Z 225.228,A -85,B 0,C 180,E1 -6111.855,E2 -6111.855} C_VEL
LIN {X 0,Y 495.853,Z 225.218,A -85,B 0,C 180,E1 -6114.309,E2 -6114.309} C_VEL
LIN {X 0,Y 495.979,Z 225.2,A -85,B 0,C 180,E1 -6117.567,E2 -6117.567} C_VEL
LIN {X 0,Y 495.927,Z 225.206,A -85,B 0,C 180,E1 -6120.815,E2 -6120.815} C_VEL
LIN {X 0,Y 495.98,Z 225.204,A -85,B 0,C 180,E1 -6122.439,E2 -6122.439} C_VEL
LIN {X 0,Y 495.862,Z 225.214,A -85,B 0,C 180,E1 -6125.697,E2 -6125.697} C_VEL
LIN {X 0,Y 495.82,Z 225.223,A -85,B 0,C 180,E1 -6128.152,E2 -6128.152} C_VEL
LIN {X 0,Y 495.859,Z 225.213,A -85,B 0,C 180,E1 -6131.448,E2 -6131.448} C_VEL
LIN {X 0,Y 495.79,Z 225.229,A -85,B 0,C 180,E1 -6134.786,E2 -6134.786} C_VEL
LIN {X 0,Y 495.768,Z 225.226,A -85,B 0,C 180,E1 -6137.322,E2 -6137.322} C_VEL
LIN {X 0,Y 495.773,Z 225.224,A -85,B 0,C 180,E1 -6139.893,E2 -6139.893} C_VEL
LIN {X 0,Y 495.771,Z 225.233,A -85,B 0,C 180,E1 -6142.862,E2 -6142.862} C_VEL
LIN {X 0,Y 495.731,Z 225.229,A -85,B 0,C 180,E1 -6146.074,E2 -6146.074} C_VEL
LIN {X 0,Y 495.741,Z 225.233,A -85,B 0,C 180,E1 -6148.819,E2 -6148.819} C_VEL
LIN {X 0,Y 495.764,Z 225.227,A -85,B 0,C 180,E1 -6151.725,E2 -6151.725} C_VEL
LIN {X 0,Y 495.771,Z 225.225,A -85,B 0,C 180,E1 -6154.693,E2 -6154.693} C_VEL
LIN {X 0,Y 495.734,Z 225.235,A -85,B 0,C 180,E1 -6157.563,E2 -6157.563} C_VEL
LIN {X 0,Y 495.758,Z 225.227,A -85,B 0,C 180,E1 -6160.046,E2 -6160.046} C_VEL
LIN {X 0,Y 495.709,Z 225.233,A -85,B 0,C 180,E1 -6162.887,E2 -6162.887} C_VEL
LIN {X 0,Y 495.736,Z 225.232,A -85,B 0,C 180,E1 -6165.998,E2 -6165.998} C_VEL
LIN {X 0,Y 495.741,Z 225.23,A -85,B 0,C 180,E1 -6169.296,E2 -6169.296} C_VEL
LIN {X 0,Y 495.758,Z 225.229,A -85,B 0,C 180,E1 -6171.408,E2 -6171.408} C_VEL
LIN {X 0,Y 495.757,Z 225.228,A -85,B 0,C 180,E1 -6174.462,E2 -6174.462} C_VEL
LIN {X 0,Y 495.78,Z 225.224,A -85,B 0,C 180,E1 -6177.405,E2 -6177.405} C_VEL
LIN {X 0,Y 495.775,Z 225.232,A -85,B 0,C 180,E1 -6180.253,E2 -6180.253} C_VEL
LIN {X 0,Y 495.787,Z 225.226,A -85,B 0,C 180,E1 -6183.262,E2 -6183.262} C_VEL
LIN {X 0,Y 495.836,Z 225.351,A -85,B 0,C 180,E1 -6185.895,E2 -6185.895} C_VEL
LIN {X 0,Y 497.345,Z 234.019,A -85,B 0,C 180,E1 -6187.57,E2 -6187.57} C_VEL
LIN {X 0,Y 496.966,Z 247.36,A -85,B 0,C 180,E1 -6189.943,E2 -6189.943} C_VEL
LIN {X 0,Y 496.485,Z 263.072,A -85,B 0,C 180,E1 -6192.705,E2 -6192.705} C_VEL
LIN {X 0,Y 496.323,Z 270.458,A -85,B 0,C 180,E1 -6193.954,E2 -6193.954} C_VEL
LIN {X 0,Y 497.587,Z 278.418,A -85,B 0,C 180,E1 -6194.145,E2 -6194.145} C_VEL
LIN {X 0,Y 498.531,Z 284.581,A -85,B 0,C 180,E1 -6194.265,E2 -6194.265} C_VEL
LIN {X 0,Y 497.973,Z 378.495,A -85,B 0,C 180,E1 -6195.648,E2 -6195.648} C_VEL
LIN {X 0,Y 497.693,Z 391.657,A -85,B 0,C 180,E1 -6196.005,E2 -6196.005} C_VEL
LIN {X 0,Y 497.33,Z 404.332,A -85,B 0,C 180,E1 -6196.515,E2 -6196.515} C_VEL
LIN {X 0,Y 496.999,Z 416.557,A -85,B 0,C 180,E1 -6197.193,E2 -6197.193} C_VEL
LIN {X 0,Y 496.672,Z 427.247,A -85,B 0,C 180,E1 -6197.952,E2 -6197.952} C_VEL
LIN {X 0,Y 496.265,Z 437.723,A -85,B 0,C 180,E1 -6198.874,E2 -6198.874} C_VEL
LIN {X 0,Y 495.916,Z 446.285,A -85,B 0,C 180,E1 -6199.795,E2 -6199.795} C_VEL
LIN {X 0,Y 495.613,Z 454.179,A -85,B 0,C 180,E1 -6200.819,E2 -6200.819} C_VEL
LIN {X 0,Y 495.373,Z 461.883,A -85,B 0,C 180,E1 -6202.048,E2 -6202.048} C_VEL
LIN {X 0,Y 495.171,Z 468.975,A -85,B 0,C 180,E1 -6203.479,E2 -6203.479} C_VEL
LIN {X 0,Y 495.116,Z 473.693,A -85,B 0,C 180,E1 -6204.705,E2 -6204.705} C_VEL
LIN {X 0,Y 495.035,Z 477.297,A -85,B 0,C 180,E1 -6205.928,E2 -6205.928} C_VEL
LIN {X 0,Y 495.044,Z 479.157,A -85,B 0,C 180,E1 -6206.743,E2 -6206.743} C_VEL
LIN {X 0,Y 494.963,Z 481.543,A -85,B 0,C 180,E1 -6208.371,E2 -6208.371} C_VEL
LIN {X 0,Y 494.9,Z 482.365,A -85,B 0,C 180,E1 -6209.999,E2 -6209.999} C_VEL
LIN {X 0,Y 494.962,Z 481.543,A -85,B 0,C 180,E1 -6211.626,E2 -6211.626} C_VEL
LIN {X 0,Y 495.043,Z 479.156,A -85,B 0,C 180,E1 -6213.254,E2 -6213.254} C_VEL
LIN {X 0,Y 495.009,Z 476.223,A -85,B 0,C 180,E1 -6214.477,E2 -6214.477} C_VEL
LIN {X 0,Y 495.146,Z 472.255,A -85,B 0,C 180,E1 -6215.701,E2 -6215.701} C_VEL
LIN {X 0,Y 495.242,Z 466.147,A -85,B 0,C 180,E1 -6217.132,E2 -6217.132} C_VEL
LIN {X 0,Y 495.452,Z 459.478,A -85,B 0,C 180,E1 -6218.359,E2 -6218.359} C_VEL
LIN {X 0,Y 495.726,Z 451.204,A -85,B 0,C 180,E1 -6219.588,E2 -6219.588} C_VEL
LIN {X 0,Y 496.003,Z 442.719,A -85,B 0,C 180,E1 -6220.613,E2 -6220.613} C_VEL
LIN {X 0,Y 496.471,Z 432.236,A -85,B 0,C 180,E1 -6221.636,E2 -6221.636} C_VEL
LIN {X 0,Y 496.797,Z 421.569,A -85,B 0,C 180,E1 -6222.479,E2 -6222.479} C_VEL
LIN {X 0,Y 497.198,Z 410.49,A -85,B 0,C 180,E1 -6223.174,E2 -6223.174} C_VEL
LIN {X 0,Y 497.538,Z 398.804,A -85,B 0,C 180,E1 -6223.737,E2 -6223.737} C_VEL
LIN {X 0,Y 497.805,Z 385.345,A -85,B 0,C 180,E1 -6224.198,E2 -6224.198} C_VEL
LIN {X 0,Y 498.092,Z 371.998,A -85,B 0,C 180,E1 -6224.477,E2 -6224.477} C_VEL
LIN {X 0,Y 498.434,Z 283.449,A -85,B 0,C 180,E1 -6225.772,E2 -6225.772} C_VEL
LIN {X 0,Y 496.331,Z 270.71,A -85,B 0,C 180,E1 -6226.043,E2 -6226.043} C_VEL
LIN {X 0,Y 496.301,Z 269.606,A -85,B 0,C 180,E1 -6226.165,E2 -6226.165} C_VEL
LIN {X 0,Y 496.809,Z 252.09,A -85,B 0,C 180,E1 -6229.201,E2 -6229.201} C_VEL
LIN {X 0,Y 497.429,Z 235.07,A -85,B 0,C 180,E1 -6232.205,E2 -6232.205} C_VEL
LIN {X 0,Y 495.849,Z 225.467,A -85,B 0,C 180,E1 -6234.046,E2 -6234.046} C_VEL
LIN {X 0,Y 495.738,Z 225.235,A -85,B 0,C 180,E1 -6235.168,E2 -6235.168} C_VEL
LIN {X 0,Y 495.779,Z 225.233,A -85,B 0,C 180,E1 -6237.89,E2 -6237.89} C_VEL
LIN {X 0,Y 495.752,Z 225.228,A -85,B 0,C 180,E1 -6240.685,E2 -6240.685} C_VEL
LIN {X 0,Y 495.76,Z 225.229,A -85,B 0,C 180,E1 -6243.562,E2 -6243.562} C_VEL
LIN {X 0,Y 495.716,Z 225.235,A -85,B 0,C 180,E1 -6246.543,E2 -6246.543} C_VEL
LIN {X 0,Y 495.751,Z 225.229,A -85,B 0,C 180,E1 -6249.636,E2 -6249.636} C_VEL
LIN {X 0,Y 495.734,Z 225.233,A -85,B 0,C 180,E1 -6252.504,E2 -6252.504} C_VEL
LIN {X 0,Y 495.736,Z 225.228,A -85,B 0,C 180,E1 -6255.139,E2 -6255.139} C_VEL
LIN {X 0,Y 495.743,Z 225.231,A -85,B 0,C 180,E1 -6258.215,E2 -6258.215} C_VEL
LIN {X 0,Y 495.743,Z 225.228,A -85,B 0,C 180,E1 -6261.405,E2 -6261.405} C_VEL
LIN {X 0,Y 495.742,Z 225.234,A -85,B 0,C 180,E1 -6264.46,E2 -6264.46} C_VEL
LIN {X 0,Y 495.764,Z 225.224,A -85,B 0,C 180,E1 -6267.403,E2 -6267.403} C_VEL
LIN {X 0,Y 495.757,Z 225.229,A -85,B 0,C 180,E1 -6270.251,E2 -6270.251} C_VEL
LIN {X 0,Y 495.735,Z 225.231,A -85,B 0,C 180,E1 -6273.267,E2 -6273.267} C_VEL
LIN {X 0,Y 495.732,Z 225.234,A -85,B 0,C 180,E1 -6276.609,E2 -6276.609} C_VEL
LIN {X 0,Y 495.772,Z 225.227,A -85,B 0,C 180,E1 -6279.321,E2 -6279.321} C_VEL
LIN {X 0,Y 495.771,Z 225.224,A -85,B 0,C 180,E1 -6281.826,E2 -6281.826} C_VEL
LIN {X 0,Y 495.767,Z 225.233,A -85,B 0,C 180,E1 -6285.214,E2 -6285.214} C_VEL
LIN {X 0,Y 495.838,Z 225.214,A -85,B 0,C 180,E1 -6288.552,E2 -6288.552} C_VEL
LIN {X 0,Y 495.804,Z 225.218,A -85,B 0,C 180,E1 -6291.848,E2 -6291.848} C_VEL
LIN {X 0,Y 495.861,Z 225.213,A -85,B 0,C 180,E1 -6294.303,E2 -6294.303} C_VEL
LIN {X 0,Y 495.957,Z 225.207,A -85,B 0,C 180,E1 -6297.56,E2 -6297.56} C_VEL
LIN {X 0,Y 495.95,Z 225.203,A -85,B 0,C 180,E1 -6299.997,E2 -6299.997} C_VEL
LIN {X 0,Y 495.957,Z 225.201,A -85,B 0,C 180,E1 -6302.433,E2 -6302.433} C_VEL
LIN {X 0,Y 495.832,Z 225.222,A -85,B 0,C 180,E1 -6305.691,E2 -6305.691} C_VEL
LIN {X 0,Y 495.81,Z 225.222,A -85,B 0,C 180,E1 -6308.145,E2 -6308.145} C_VEL
LIN {X 0,Y 495.83,Z 225.221,A -85,B 0,C 180,E1 -6311.442,E2 -6311.442} C_VEL
LIN {X 0,Y 495.758,Z 225.227,A -85,B 0,C 180,E1 -6314.78,E2 -6314.78} C_VEL
LIN {X 0,Y 495.73,Z 225.229,A -85,B 0,C 180,E1 -6317.317,E2 -6317.317} C_VEL
LIN {X 0,Y 495.743,Z 225.234,A -85,B 0,C 180,E1 -6319.887,E2 -6319.887} C_VEL
LIN {X 0,Y 495.732,Z 225.23,A -85,B 0,C 180,E1 -6322.857,E2 -6322.857} C_VEL
LIN {X 0,Y 495.751,Z 225.232,A -85,B 0,C 180,E1 -6326.065,E2 -6326.065} C_VEL
LIN {X 0,Y 495.741,Z 225.229,A -85,B 0,C 180,E1 -6328.812,E2 -6328.812} C_VEL
LIN {X 0,Y 495.724,Z 225.232,A -85,B 0,C 180,E1 -6331.723,E2 -6331.723} C_VEL
LIN {X 0,Y 495.744,Z 225.233,A -85,B 0,C 180,E1 -6334.693,E2 -6334.693} C_VEL
LIN {X 0,Y 495.699,Z 225.235,A -85,B 0,C 180,E1 -6337.559,E2 -6337.559} C_VEL
LIN {X 0,Y 495.758,Z 225.23,A -85,B 0,C 180,E1 -6340.05,E2 -6340.05} C_VEL
LIN {X 0,Y 495.727,Z 225.239,A -85,B 0,C 180,E1 -6342.877,E2 -6342.877} C_VEL
LIN {X 0,Y 495.697,Z 225.239,A -85,B 0,C 180,E1 -6345.997,E2 -6345.997} C_VEL
LIN {X 0,Y 495.777,Z 225.428,A -85,B 0,C 180,E1 -6347.051,E2 -6347.051} C_VEL
LIN {X 0,Y 496.867,Z 231.925,A -85,B 0,C 180,E1 -6348.335,E2 -6348.335} C_VEL
LIN {X 0,Y 496.478,Z 247.086,A -85,B 0,C 180,E1 -6351.121,E2 -6351.121} C_VEL
LIN {X 0,Y 496.296,Z 257.395,A -85,B 0,C 180,E1 -6352.967,E2 -6352.967} C_VEL
LIN {X 0,Y 496.917,Z 261.042,A -85,B 0,C 180,E1 -6353.084,E2 -6353.084} C_VEL
LIN {X 0,Y 498.611,Z 271.308,A -85,B 0,C 180,E1 -6353.294,E2 -6353.294} C_VEL
LIN {X 0,Y 498.324,Z 313.871,A -85,B 0,C 180,E1 -6353.914,E2 -6353.914} C_VEL
LIN {X 0,Y 497.611,Z 319.713,A -85,B 0,C 180,E1 -6353.977,E2 -6353.977} C_VEL
LIN {X 0,Y 491.965,Z 338.701,A -85,B 0,C 180,E1 -6354.08,E2 -6354.08} C_VEL
LIN {X 0,Y 491.325,Z 344.54,A -85,B 0,C 180,E1 -6354.147,E2 -6354.147} C_VEL
LIN {X 0,Y 491.141,Z 366.914,A -85,B 0,C 180,E1 -6354.512,E2 -6354.512} C_VEL
LIN {X 0,Y 490.839,Z 380.19,A -85,B 0,C 180,E1 -6354.898,E2 -6354.898} C_VEL
LIN {X 0,Y 490.55,Z 392.143,A -85,B 0,C 180,E1 -6355.412,E2 -6355.412} C_VEL
LIN {X 0,Y 490.158,Z 404.012,A -85,B 0,C 180,E1 -6356.096,E2 -6356.096} C_VEL
LIN {X 0,Y 489.674,Z 415.602,A -85,B 0,C 180,E1 -6356.95,E2 -6356.95} C_VEL
LIN {X 0,Y 489.294,Z 426.057,A -85,B 0,C 180,E1 -6357.926,E2 -6357.926} C_VEL
LIN {X 0,Y 488.897,Z 435.805,A -85,B 0,C 180,E1 -6359.056,E2 -6359.056} C_VEL
LIN {X 0,Y 488.539,Z 444.127,A -85,B 0,C 180,E1 -6360.246,E2 -6360.246} C_VEL
LIN {X 0,Y 488.357,Z 450.538,A -85,B 0,C 180,E1 -6361.374,E2 -6361.374} C_VEL
LIN {X 0,Y 488.165,Z 456.066,A -85,B 0,C 180,E1 -6362.57,E2 -6362.57} C_VEL
LIN {X 0,Y 488.046,Z 461.034,A -85,B 0,C 180,E1 -6363.948,E2 -6363.948} C_VEL
LIN {X 0,Y 487.915,Z 464.656,A -85,B 0,C 180,E1 -6365.311,E2 -6365.311} C_VEL
LIN {X 0,Y 487.81,Z 466.404,A -85,B 0,C 180,E1 -6366.211,E2 -6366.211} C_VEL
LIN {X 0,Y 487.769,Z 467.783,A -85,B 0,C 180,E1 -6367.227,E2 -6367.227} C_VEL
LIN {X 0,Y 487.753,Z 468.731,A -85,B 0,C 180,E1 -6368.888,E2 -6368.888} C_VEL
LIN {X 0,Y 487.804,Z 468.592,A -85,B 0,C 180,E1 -6369.772,E2 -6369.772} C_VEL
LIN {X 0,Y 487.8,Z 467.974,A -85,B 0,C 180,E1 -6370.649,E2 -6370.649} C_VEL
LIN {X 0,Y 487.829,Z 466.267,A -85,B 0,C 180,E1 -6371.943,E2 -6371.943} C_VEL
LIN {X 0,Y 487.965,Z 462.345,A -85,B 0,C 180,E1 -6373.69,E2 -6373.69} C_VEL
LIN {X 0,Y 488.111,Z 458.117,A -85,B 0,C 180,E1 -6374.981,E2 -6374.981} C_VEL
LIN {X 0,Y 488.273,Z 451.649,A -85,B 0,C 180,E1 -6376.475,E2 -6376.475} C_VEL
LIN {X 0,Y 488.57,Z 443.947,A -85,B 0,C 180,E1 -6377.853,E2 -6377.853} C_VEL
LIN {X 0,Y 488.85,Z 435.765,A -85,B 0,C 180,E1 -6379.02,E2 -6379.02} C_VEL
LIN {X 0,Y 489.264,Z 425.718,A -85,B 0,C 180,E1 -6380.18,E2 -6380.18} C_VEL
LIN {X 0,Y 489.641,Z 415.507,A -85,B 0,C 180,E1 -6381.125,E2 -6381.125} C_VEL
LIN {X 0,Y 490.07,Z 405.185,A -85,B 0,C 180,E1 -6381.895,E2 -6381.895} C_VEL
LIN {X 0,Y 490.464,Z 393.354,A -85,B 0,C 180,E1 -6382.592,E2 -6382.592} C_VEL
LIN {X 0,Y 490.787,Z 381.649,A -85,B 0,C 180,E1 -6383.113,E2 -6383.113} C_VEL
LIN {X 0,Y 491.061,Z 369.107,A -85,B 0,C 180,E1 -6383.504,E2 -6383.504} C_VEL
LIN {X 0,Y 491.196,Z 353.345,A -85,B 0,C 180,E1 -6383.79,E2 -6383.79} C_VEL
LIN {X 0,Y 491.538,Z 270.419,A -85,B 0,C 180,E1 -6385.016,E2 -6385.016} C_VEL
LIN {X 0,Y 489.341,Z 258.147,A -85,B 0,C 180,E1 -6385.29,E2 -6385.29} C_VEL
LIN {X 0,Y 489.282,Z 256.735,A -85,B 0,C 180,E1 -6385.47,E2 -6385.47} C_VEL
LIN {X 0,Y 489.794,Z 242.762,A -85,B 0,C 180,E1 -6388.151,E2 -6388.151} C_VEL
LIN {X 0,Y 490.04,Z 233.275,A -85,B 0,C 180,E1 -6390.001,E2 -6390.001} C_VEL
LIN {X 0,Y 488.801,Z 226.166,A -85,B 0,C 180,E1 -6391.52,E2 -6391.52} C_VEL
LIN {X 0,Y 488.916,Z 226.084,A -85,B 0,C 180,E1 -6392.473,E2 -6392.473} C_VEL
LIN {X 0,Y 488.812,Z 226.098,A -85,B 0,C 180,E1 -6395.777,E2 -6395.777} C_VEL
LIN {X 0,Y 488.774,Z 226.096,A -85,B 0,C 180,E1 -6398.268,E2 -6398.268} C_VEL
LIN {X 0,Y 488.787,Z 226.103,A -85,B 0,C 180,E1 -6401.614,E2 -6401.614} C_VEL
LIN {X 0,Y 488.719,Z 226.103,A -85,B 0,C 180,E1 -6405.003,E2 -6405.003} C_VEL
LIN {X 0,Y 488.716,Z 226.104,A -85,B 0,C 180,E1 -6408.445,E2 -6408.445} C_VEL
LIN {X 0,Y 488.668,Z 226.109,A -85,B 0,C 180,E1 -6411.074,E2 -6411.074} C_VEL
LIN {X 0,Y 488.636,Z 226.118,A -85,B 0,C 180,E1 -6413.75,E2 -6413.75} C_VEL
LIN {X 0,Y 488.678,Z 226.108,A -85,B 0,C 180,E1 -6416.929,E2 -6416.929} C_VEL
LIN {X 0,Y 488.69,Z 226.115,A -85,B 0,C 180,E1 -6420.223,E2 -6420.223} C_VEL
LIN {X 0,Y 488.677,Z 226.108,A -85,B 0,C 180,E1 -6423.483,E2 -6423.483} C_VEL
LIN {X 0,Y 488.634,Z 226.122,A -85,B 0,C 180,E1 -6426.355,E2 -6426.355} C_VEL
LIN {X 0,Y 488.658,Z 226.11,A -85,B 0,C 180,E1 -6429.26,E2 -6429.26} C_VEL
LIN {X 0,Y 488.64,Z 226.12,A -85,B 0,C 180,E1 -6432.532,E2 -6432.532} C_VEL
LIN {X 0,Y 488.677,Z 226.11,A -85,B 0,C 180,E1 -6435.201,E2 -6435.201} C_VEL
LIN {X 0,Y 488.655,Z 226.116,A -85,B 0,C 180,E1 -6438.585,E2 -6438.585} C_VEL
LIN {X 0,Y 488.678,Z 226.116,A -85,B 0,C 180,E1 -6440.953,E2 -6440.953} C_VEL
LIN {X 0,Y 488.659,Z 226.11,A -85,B 0,C 180,E1 -6443.872,E2 -6443.872} C_VEL
LIN {X 0,Y 488.687,Z 226.112,A -85,B 0,C 180,E1 -6446.879,E2 -6446.879} C_VEL
LIN {X 0,Y 488.704,Z 226.106,A -85,B 0,C 180,E1 -6449.784,E2 -6449.784} C_VEL
LIN {X 0,Y 488.686,Z 226.113,A -85,B 0,C 180,E1 -6453.083,E2 -6453.083} C_VEL
LIN {X 0,Y 488.66,Z 226.11,A -85,B 0,C 180,E1 -6456.257,E2 -6456.257} C_VEL
LIN {X 0,Y 488.741,Z 226.104,A -85,B 0,C 180,E1 -6459.18,E2 -6459.18} C_VEL
LIN {X 0,Y 488.743,Z 226.108,A -85,B 0,C 180,E1 -6461.637,E2 -6461.637} C_VEL
LIN {X 0,Y 488.754,Z 226.099,A -85,B 0,C 180,E1 -6465.003,E2 -6465.003} C_VEL
LIN {X 0,Y 488.783,Z 226.096,A -85,B 0,C 180,E1 -6468.391,E2 -6468.391} C_VEL
LIN {X 0,Y 488.762,Z 226.104,A -85,B 0,C 180,E1 -6471.736,E2 -6471.736} C_VEL
LIN {X 0,Y 488.813,Z 226.096,A -85,B 0,C 180,E1 -6474.227,E2 -6474.227} C_VEL
LIN {X 0,Y 488.945,Z 226.076,A -85,B 0,C 180,E1 -6477.532,E2 -6477.532} C_VEL
LIN {X 0,Y 488.945,Z 226.081,A -85,B 0,C 180,E1 -6480.003,E2 -6480.003} C_VEL
LIN {X 0,Y 488.946,Z 226.08,A -85,B 0,C 180,E1 -6482.475,E2 -6482.475} C_VEL
LIN {X 0,Y 488.821,Z 226.091,A -85,B 0,C 180,E1 -6485.779,E2 -6485.779} C_VEL
LIN {X 0,Y 488.767,Z 226.103,A -85,B 0,C 180,E1 -6488.27,E2 -6488.27} C_VEL
LIN {X 0,Y 488.814,Z 226.09,A -85,B 0,C 180,E1 -6491.615,E2 -6491.615} C_VEL
LIN {X 0,Y 488.767,Z 226.1,A -85,B 0,C 180,E1 -6495.003,E2 -6495.003} C_VEL
LIN {X 0,Y 488.758,Z 226.102,A -85,B 0,C 180,E1 -6498.445,E2 -6498.445} C_VEL
LIN {X 0,Y 488.72,Z 226.108,A -85,B 0,C 180,E1 -6501.073,E2 -6501.073} C_VEL
LIN {X 0,Y 488.682,Z 226.107,A -85,B 0,C 180,E1 -6503.749,E2 -6503.749} C_VEL
LIN {X 0,Y 488.712,Z 226.111,A -85,B 0,C 180,E1 -6506.923,E2 -6506.923} C_VEL
LIN {X 0,Y 488.73,Z 226.101,A -85,B 0,C 180,E1 -6510.221,E2 -6510.221} C_VEL
LIN {X 0,Y 488.724,Z 226.107,A -85,B 0,C 180,E1 -6513.481,E2 -6513.481} C_VEL
LIN {X 0,Y 488.684,Z 226.107,A -85,B 0,C 180,E1 -6516.353,E2 -6516.353} C_VEL
LIN {X 0,Y 488.708,Z 226.11,A -85,B 0,C 180,E1 -6519.256,E2 -6519.256} C_VEL
LIN {X 0,Y 488.682,Z 226.115,A -85,B 0,C 180,E1 -6521.595,E2 -6521.595} C_VEL
LIN {X 0,Y 488.715,Z 226.103,A -85,B 0,C 180,E1 -6524.803,E2 -6524.803} C_VEL
LIN {X 0,Y 488.663,Z 226.115,A -85,B 0,C 180,E1 -6527.47,E2 -6527.47} C_VEL
LIN {X 0,Y 488.718,Z 226.11,A -85,B 0,C 180,E1 -6529.674,E2 -6529.674} C_VEL
LIN {X 0,Y 488.682,Z 226.107,A -85,B 0,C 180,E1 -6532.84,E2 -6532.84} C_VEL
LIN {X 0,Y 488.742,Z 226.107,A -85,B 0,C 180,E1 -6535.887,E2 -6535.887} C_VEL
LIN {X 0,Y 488.703,Z 226.105,A -85,B 0,C 180,E1 -6538.82,E2 -6538.82} C_VEL
LIN {X 0,Y 488.725,Z 226.107,A -85,B 0,C 180,E1 -6541.669,E2 -6541.669} C_VEL
LIN {X 0,Y 488.718,Z 226.112,A -85,B 0,C 180,E1 -6544.441,E2 -6544.441} C_VEL
LIN {X 0,Y 488.75,Z 226.193,A -85,B 0,C 180,E1 -6545.693,E2 -6545.693} C_VEL
LIN {X 0,Y 490.358,Z 235.085,A -85,B 0,C 180,E1 -6547.455,E2 -6547.455} C_VEL
LIN {X 0,Y 490.118,Z 244.79,A -85,B 0,C 180,E1 -6549.212,E2 -6549.212} C_VEL
LIN {X 0,Y 489.572,Z 261.726,A -85,B 0,C 180,E1 -6552.238,E2 -6552.238} C_VEL
LIN {X 0,Y 489.322,Z 270.234,A -85,B 0,C 180,E1 -6553.712,E2 -6553.712} C_VEL
LIN {X 0,Y 489.957,Z 274.75,A -85,B 0,C 180,E1 -6553.847,E2 -6553.847} C_VEL
LIN {X 0,Y 491.679,Z 285.627,A -85,B 0,C 180,E1 -6554.065,E2 -6554.065} C_VEL
LIN {X 0,Y 491.093,Z 378.103,A -85,B 0,C 180,E1 -6555.442,E2 -6555.442} C_VEL
LIN {X 0,Y 490.779,Z 391.36,A -85,B 0,C 180,E1 -6555.803,E2 -6555.803} C_VEL
LIN {X 0,Y 490.427,Z 404.086,A -85,B 0,C 180,E1 -6556.322,E2 -6556.322} C_VEL
LIN {X 0,Y 490.103,Z 415.244,A -85,B 0,C 180,E1 -6556.936,E2 -6556.936} C_VEL
LIN {X 0,Y 489.7,Z 427.064,A -85,B 0,C 180,E1 -6557.778,E2 -6557.778} C_VEL
LIN {X 0,Y 489.279,Z 437.556,A -85,B 0,C 180,E1 -6558.713,E2 -6558.713} C_VEL
LIN {X 0,Y 488.878,Z 446.129,A -85,B 0,C 180,E1 -6559.647,E2 -6559.647} C_VEL
LIN {X 0,Y 488.566,Z 454.034,A -85,B 0,C 180,E1 -6560.686,E2 -6560.686} C_VEL
LIN {X 0,Y 488.326,Z 461.754,A -85,B 0,C 180,E1 -6561.932,E2 -6561.932} C_VEL
LIN {X 0,Y 488.104,Z 468.856,A -85,B 0,C 180,E1 -6563.384,E2 -6563.384} C_VEL
LIN {X 0,Y 488.049,Z 473.582,A -85,B 0,C 180,E1 -6564.628,E2 -6564.628} C_VEL
LIN {X 0,Y 487.93,Z 477.191,A -85,B 0,C 180,E1 -6565.869,E2 -6565.869} C_VEL
LIN {X 0,Y 487.967,Z 479.053,A -85,B 0,C 180,E1 -6566.696,E2 -6566.696} C_VEL
LIN {X 0,Y 487.89,Z 481.443,A -85,B 0,C 180,E1 -6568.348,E2 -6568.348} C_VEL
LIN {X 0,Y 487.821,Z 482.267,A -85,B 0,C 180,E1 -6569.999,E2 -6569.999} C_VEL
LIN {X 0,Y 487.89,Z 481.446,A -85,B 0,C 180,E1 -6571.65,E2 -6571.65} C_VEL
LIN {X 0,Y 487.966,Z 479.061,A -85,B 0,C 180,E1 -6573.301,E2 -6573.301} C_VEL
LIN {X 0,Y 487.922,Z 476.13,A -85,B 0,C 180,E1 -6574.542,E2 -6574.542} C_VEL
LIN {X 0,Y 488.063,Z 472.165,A -85,B 0,C 180,E1 -6575.784,E2 -6575.784} C_VEL
LIN {X 0,Y 488.132,Z 467.062,A -85,B 0,C 180,E1 -6577.028,E2 -6577.028} C_VEL
LIN {X 0,Y 488.343,Z 460.635,A -85,B 0,C 180,E1 -6578.273,E2 -6578.273} C_VEL
LIN {X 0,Y 488.621,Z 452.619,A -85,B 0,C 180,E1 -6579.52,E2 -6579.52} C_VEL
LIN {X 0,Y 488.94,Z 444.45,A -85,B 0,C 180,E1 -6580.559,E2 -6580.559} C_VEL
LIN {X 0,Y 489.369,Z 434.487,A -85,B 0,C 180,E1 -6581.597,E2 -6581.597} C_VEL
LIN {X 0,Y 489.774,Z 424.659,A -85,B 0,C 180,E1 -6582.428,E2 -6582.428} C_VEL
LIN {X 0,Y 490.161,Z 414.071,A -85,B 0,C 180,E1 -6583.15,E2 -6583.15} C_VEL
LIN {X 0,Y 490.53,Z 402.262,A -85,B 0,C 180,E1 -6583.778,E2 -6583.778} C_VEL
LIN {X 0,Y 490.889,Z 388.948,A -85,B 0,C 180,E1 -6584.297,E2 -6584.297} C_VEL
LIN {X 0,Y 491.185,Z 376.637,A -85,B 0,C 180,E1 -6584.605,E2 -6584.605} C_VEL
LIN {X 0,Y 491.731,Z 284.97,A -85,B 0,C 180,E1 -6585.973,E2 -6585.973} C_VEL
LIN {X 0,Y 489.311,Z 270.255,A -85,B 0,C 180,E1 -6586.306,E2 -6586.306} C_VEL
LIN {X 0,Y 489.771,Z 255.222,A -85,B 0,C 180,E1 -6588.918,E2 -6588.918} C_VEL
LIN {X 0,Y 490.493,Z 236.248,A -85,B 0,C 180,E1 -6592.314,E2 -6592.314} C_VEL
LIN {X 0,Y 488.796,Z 226.34,A -85,B 0,C 180,E1 -6594.246,E2 -6594.246} C_VEL
LIN {X 0,Y 488.706,Z 226.111,A -85,B 0,C 180,E1 -6595.04,E2 -6595.04} C_VEL
LIN {X 0,Y 488.734,Z 226.107,A -85,B 0,C 180,E1 -6597.396,E2 -6597.396} C_VEL
LIN {X 0,Y 488.71,Z 226.107,A -85,B 0,C 180,E1 -6600.36,E2 -6600.36} C_VEL
LIN {X 0,Y 488.736,Z 226.103,A -85,B 0,C 180,E1 -6603.482,E2 -6603.482} C_VEL
LIN {X 0,Y 488.674,Z 226.114,A -85,B 0,C 180,E1 -6606.351,E2 -6606.351} C_VEL
LIN {X 0,Y 488.697,Z 226.105,A -85,B 0,C 180,E1 -6609.253,E2 -6609.253} C_VEL
LIN {X 0,Y 488.697,Z 226.107,A -85,B 0,C 180,E1 -6611.596,E2 -6611.596} C_VEL
LIN {X 0,Y 488.7,Z 226.107,A -85,B 0,C 180,E1 -6614.8,E2 -6614.8} C_VEL
LIN {X 0,Y 488.687,Z 226.103,A -85,B 0,C 180,E1 -6617.472,E2 -6617.472} C_VEL
LIN {X 0,Y 488.691,Z 226.111,A -85,B 0,C 180,E1 -6620.743,E2 -6620.743} C_VEL
LIN {X 0,Y 488.666,Z 226.109,A -85,B 0,C 180,E1 -6623.865,E2 -6623.865} C_VEL
LIN {X 0,Y 488.735,Z 226.104,A -85,B 0,C 180,E1 -6626.875,E2 -6626.875} C_VEL
LIN {X 0,Y 488.717,Z 226.103,A -85,B 0,C 180,E1 -6629.778,E2 -6629.778} C_VEL
LIN {X 0,Y 488.695,Z 226.11,A -85,B 0,C 180,E1 -6633.075,E2 -6633.075} C_VEL
LIN {X 0,Y 488.662,Z 226.111,A -85,B 0,C 180,E1 -6636.25,E2 -6636.25} C_VEL
LIN {X 0,Y 488.74,Z 226.105,A -85,B 0,C 180,E1 -6639.173,E2 -6639.173} C_VEL
LIN {X 0,Y 488.74,Z 226.101,A -85,B 0,C 180,E1 -6641.629,E2 -6641.629} C_VEL
LIN {X 0,Y 488.744,Z 226.106,A -85,B 0,C 180,E1 -6644.996,E2 -6644.996} C_VEL
LIN {X 0,Y 488.793,Z 226.091,A -85,B 0,C 180,E1 -6648.384,E2 -6648.384} C_VEL
LIN {X 0,Y 488.75,Z 226.098,A -85,B 0,C 180,E1 -6651.73,E2 -6651.73} C_VEL
LIN {X 0,Y 488.819,Z 226.091,A -85,B 0,C 180,E1 -6654.221,E2 -6654.221} C_VEL
LIN {X 0,Y 488.924,Z 226.082,A -85,B 0,C 180,E1 -6657.525,E2 -6657.525} C_VEL
LIN {X 0,Y 488.92,Z 226.079,A -85,B 0,C 180,E1 -6659.997,E2 -6659.997} C_VEL
LIN {X 0,Y 488.924,Z 226.077,A -85,B 0,C 180,E1 -6662.468,E2 -6662.468} C_VEL
LIN {X 0,Y 488.792,Z 226.099,A -85,B 0,C 180,E1 -6665.773,E2 -6665.773} C_VEL
LIN {X 0,Y 488.76,Z 226.099,A -85,B 0,C 180,E1 -6668.264,E2 -6668.264} C_VEL
LIN {X 0,Y 488.784,Z 226.101,A -85,B 0,C 180,E1 -6671.609,E2 -6671.609} C_VEL
LIN {X 0,Y 488.733,Z 226.102,A -85,B 0,C 180,E1 -6674.997,E2 -6674.997} C_VEL
LIN {X 0,Y 488.721,Z 226.106,A -85,B 0,C 180,E1 -6678.439,E2 -6678.439} C_VEL
LIN {X 0,Y 488.681,Z 226.108,A -85,B 0,C 180,E1 -6681.068,E2 -6681.068} C_VEL
LIN {X 0,Y 488.649,Z 226.114,A -85,B 0,C 180,E1 -6683.743,E2 -6683.743} C_VEL
LIN {X 0,Y 488.763,Z 226.099,A -85,B 0,C 180,E1 -6686.941,E2 -6686.941} C_VEL
LIN {X 0,Y 488.679,Z 226.115,A -85,B 0,C 180,E1 -6690.36,E2 -6690.36} C_VEL
LIN {X 0,Y 488.703,Z 226.105,A -85,B 0,C 180,E1 -6693.482,E2 -6693.482} C_VEL
LIN {X 0,Y 488.656,Z 226.114,A -85,B 0,C 180,E1 -6696.353,E2 -6696.353} C_VEL
LIN {X 0,Y 488.714,Z 226.108,A -85,B 0,C 180,E1 -6699.247,E2 -6699.247} C_VEL
LIN {X 0,Y 488.697,Z 226.112,A -85,B 0,C 180,E1 -6702.519,E2 -6702.519} C_VEL
LIN {X 0,Y 488.674,Z 226.116,A -85,B 0,C 180,E1 -6705.196,E2 -6705.196} C_VEL
LIN {X 0,Y 488.687,Z 226.216,A -85,B 0,C 180,E1 -6706.831,E2 -6706.831} C_VEL
LIN {X 0,Y 489.924,Z 233.072,A -85,B 0,C 180,E1 -6708.233,E2 -6708.233} C_VEL
LIN {X 0,Y 489.488,Z 248.426,A -85,B 0,C 180,E1 -6711.088,E2 -6711.088} C_VEL
LIN {X 0,Y 489.318,Z 257.524,A -85,B 0,C 180,E1 -6712.732,E2 -6712.732} C_VEL
LIN {X 0,Y 490.384,Z 263.336,A -85,B 0,C 180,E1 -6712.894,E2 -6712.894} C_VEL
LIN {X 0,Y 491.806,Z 271.899,A -85,B 0,C 180,E1 -6713.073,E2 -6713.073} C_VEL
LIN {X 0,Y 491.325,Z 344.54,A -85,B 0,C 180,E1 -6714.147,E2 -6714.147} C_VEL
LIN {X 0,Y 490.639,Z 350.391,A -85,B 0,C 180,E1 -6714.21,E2 -6714.21} C_VEL
LIN {X 0,Y 484.96,Z 368.348,A -85,B 0,C 180,E1 -6714.351,E2 -6714.351} C_VEL
LIN {X 0,Y 484.177,Z 373.124,A -85,B 0,C 180,E1 -6714.456,E2 -6714.456} C_VEL
LIN {X 0,Y 484.125,Z 375.037,A -85,B 0,C 180,E1 -6714.512,E2 -6714.512} C_VEL
LIN {X 0,Y 483.763,Z 387.477,A -85,B 0,C 180,E1 -6714.983,E2 -6714.983} C_VEL
LIN {X 0,Y 483.371,Z 399.61,A -85,B 0,C 180,E1 -6715.618,E2 -6715.618} C_VEL
LIN {X 0,Y 482.894,Z 411.464,A -85,B 0,C 180,E1 -6716.426,E2 -6716.426} C_VEL
LIN {X 0,Y 482.45,Z 422.474,A -85,B 0,C 180,E1 -6717.387,E2 -6717.387} C_VEL
LIN {X 0,Y 482.017,Z 432.398,A -85,B 0,C 180,E1 -6718.463,E2 -6718.463} C_VEL
LIN {X 0,Y 481.681,Z 440.809,A -85,B 0,C 180,E1 -6719.584,E2 -6719.584} C_VEL
LIN {X 0,Y 481.384,Z 447.803,A -85,B 0,C 180,E1 -6720.722,E2 -6720.722} C_VEL
LIN {X 0,Y 481.136,Z 454.73,A -85,B 0,C 180,E1 -6722.134,E2 -6722.134} C_VEL
LIN {X 0,Y 480.981,Z 460.067,A -85,B 0,C 180,E1 -6723.536,E2 -6723.536} C_VEL
LIN {X 0,Y 480.843,Z 464.14,A -85,B 0,C 180,E1 -6724.972,E2 -6724.972} C_VEL
LIN {X 0,Y 480.743,Z 465.942,A -85,B 0,C 180,E1 -6725.839,E2 -6725.839} C_VEL
LIN {X 0,Y 480.686,Z 467.767,A -85,B 0,C 180,E1 -6727.075,E2 -6727.075} C_VEL
LIN {X 0,Y 480.653,Z 468.769,A -85,B 0,C 180,E1 -6728.561,E2 -6728.561} C_VEL
LIN {X 0,Y 480.698,Z 468.776,A -85,B 0,C 180,E1 -6729.46,E2 -6729.46} C_VEL
LIN {X 0,Y 480.691,Z 468.359,A -85,B 0,C 180,E1 -6730.352,E2 -6730.352} C_VEL
LIN {X 0,Y 480.737,Z 466.618,A -85,B 0,C 180,E1 -6731.833,E2 -6731.833} C_VEL
LIN {X 0,Y 480.837,Z 463.256,A -85,B 0,C 180,E1 -6733.442,E2 -6733.442} C_VEL
LIN {X 0,Y 480.989,Z 459.307,A -85,B 0,C 180,E1 -6734.753,E2 -6734.753} C_VEL
LIN {X 0,Y 481.133,Z 454.187,A -85,B 0,C 180,E1 -6736.055,E2 -6736.055} C_VEL
LIN {X 0,Y 481.345,Z 447.744,A -85,B 0,C 180,E1 -6737.35,E2 -6737.35} C_VEL
LIN {X 0,Y 481.683,Z 439.649,A -85,B 0,C 180,E1 -6738.642,E2 -6738.642} C_VEL
LIN {X 0,Y 482.035,Z 431.404,A -85,B 0,C 180,E1 -6739.713,E2 -6739.713} C_VEL
LIN {X 0,Y 482.454,Z 421.36,A -85,B 0,C 180,E1 -6740.781,E2 -6740.781} C_VEL
LIN {X 0,Y 482.949,Z 410.871,A -85,B 0,C 180,E1 -6741.673,E2 -6741.673} C_VEL
LIN {X 0,Y 483.382,Z 398.841,A -85,B 0,C 180,E1 -6742.482,E2 -6742.482} C_VEL
LIN {X 0,Y 483.761,Z 386.491,A -85,B 0,C 180,E1 -6743.118,E2 -6743.118} C_VEL
LIN {X 0,Y 484.086,Z 373.335,A -85,B 0,C 180,E1 -6743.593,E2 -6743.593} C_VEL
LIN {X 0,Y 484.272,Z 360.738,A -85,B 0,C 180,E1 -6743.883,E2 -6743.883} C_VEL
LIN {X 0,Y 484.778,Z 271.686,A -85,B 0,C 180,E1 -6745.22,E2 -6745.22} C_VEL
LIN {X 0,Y 482.318,Z 258.031,A -85,B 0,C 180,E1 -6745.535,E2 -6745.535} C_VEL
LIN {X 0,Y 482.494,Z 252.964,A -85,B 0,C 180,E1 -6746.452,E2 -6746.452} C_VEL
LIN {X 0,Y 483.124,Z 236.967,A -85,B 0,C 180,E1 -6749.585,E2 -6749.585} C_VEL
LIN {X 0,Y 482.701,Z 231.855,A -85,B 0,C 180,E1 -6750.627,E2 -6750.627} C_VEL
LIN {X 0,Y 481.785,Z 227.011,A -85,B 0,C 180,E1 -6751.699,E2 -6751.699} C_VEL
LIN {X 0,Y 481.698,Z 226.985,A -85,B 0,C 180,E1 -6753.347,E2 -6753.347} C_VEL
LIN {X 0,Y 481.771,Z 226.974,A -85,B 0,C 180,E1 -6755.862,E2 -6755.862} C_VEL
LIN {X 0,Y 481.719,Z 226.974,A -85,B 0,C 180,E1 -6758.39,E2 -6758.39} C_VEL
LIN {X 0,Y 481.752,Z 226.977,A -85,B 0,C 180,E1 -6761.786,E2 -6761.786} C_VEL
LIN {X 0,Y 481.701,Z 226.979,A -85,B 0,C 180,E1 -6765.227,E2 -6765.227} C_VEL
LIN {X 0,Y 481.673,Z 226.98,A -85,B 0,C 180,E1 -6768.724,E2 -6768.724} C_VEL
LIN {X 0,Y 481.607,Z 226.99,A -85,B 0,C 180,E1 -6771.398,E2 -6771.398} C_VEL
LIN {X 0,Y 481.615,Z 226.995,A -85,B 0,C 180,E1 -6774.118,E2 -6774.118} C_VEL
LIN {X 0,Y 481.65,Z 226.983,A -85,B 0,C 180,E1 -6777.128,E2 -6777.128} C_VEL
LIN {X 0,Y 481.639,Z 226.987,A -85,B 0,C 180,E1 -6779.745,E2 -6779.745} C_VEL
LIN {X 0,Y 481.619,Z 226.99,A -85,B 0,C 180,E1 -6782.679,E2 -6782.679} C_VEL
LIN {X 0,Y 481.595,Z 226.991,A -85,B 0,C 180,E1 -6785.714,E2 -6785.714} C_VEL
LIN {X 0,Y 481.603,Z 226.993,A -85,B 0,C 180,E1 -6788.867,E2 -6788.867} C_VEL
LIN {X 0,Y 481.6,Z 226.99,A -85,B 0,C 180,E1 -6791.913,E2 -6791.913} C_VEL
LIN {X 0,Y 481.629,Z 226.991,A -85,B 0,C 180,E1 -6794.462,E2 -6794.462} C_VEL
LIN {X 0,Y 481.607,Z 226.988,A -85,B 0,C 180,E1 -6797.841,E2 -6797.841} C_VEL
LIN {X 0,Y 481.646,Z 226.989,A -85,B 0,C 180,E1 -6801.145,E2 -6801.145} C_VEL
LIN {X 0,Y 481.619,Z 226.988,A -85,B 0,C 180,E1 -6804.295,E2 -6804.295} C_VEL
LIN {X 0,Y 481.637,Z 226.99,A -85,B 0,C 180,E1 -6807.328,E2 -6807.328} C_VEL
LIN {X 0,Y 481.653,Z 226.983,A -85,B 0,C 180,E1 -6810.262,E2 -6810.262} C_VEL
LIN {X 0,Y 481.648,Z 226.99,A -85,B 0,C 180,E1 -6813.111,E2 -6813.111} C_VEL
LIN {X 0,Y 481.638,Z 226.987,A -85,B 0,C 180,E1 -6815.889,E2 -6815.889} C_VEL
LIN {X 0,Y 481.697,Z 226.98,A -85,B 0,C 180,E1 -6819.032,E2 -6819.032} C_VEL
LIN {X 0,Y 481.678,Z 226.981,A -85,B 0,C 180,E1 -6822.161,E2 -6822.161} C_VEL
LIN {X 0,Y 481.737,Z 226.972,A -85,B 0,C 180,E1 -6824.78,E2 -6824.78} C_VEL
LIN {X 0,Y 481.734,Z 226.975,A -85,B 0,C 180,E1 -6828.218,E2 -6828.218} C_VEL
LIN {X 0,Y 481.721,Z 226.979,A -85,B 0,C 180,E1 -6831.615,E2 -6831.615} C_VEL
LIN {X 0,Y 481.775,Z 226.974,A -85,B 0,C 180,E1 -6834.143,E2 -6834.143} C_VEL
LIN {X 0,Y 481.911,Z 226.952,A -85,B 0,C 180,E1 -6837.496,E2 -6837.496} C_VEL
LIN {X 0,Y 481.914,Z 226.957,A -85,B 0,C 180,E1 -6840.003,E2 -6840.003} C_VEL
LIN {X 0,Y 481.912,Z 226.955,A -85,B 0,C 180,E1 -6842.511,E2 -6842.511} C_VEL
LIN {X 0,Y 481.782,Z 226.969,A -85,B 0,C 180,E1 -6845.864,E2 -6845.864} C_VEL
LIN {X 0,Y 481.726,Z 226.982,A -85,B 0,C 180,E1 -6848.392,E2 -6848.392} C_VEL
LIN {X 0,Y 481.761,Z 226.97,A -85,B 0,C 180,E1 -6851.787,E2 -6851.787} C_VEL
LIN {X 0,Y 481.751,Z 226.972,A -85,B 0,C 180,E1 -6855.227,E2 -6855.227} C_VEL
LIN {X 0,Y 481.719,Z 226.983,A -85,B 0,C 180,E1 -6858.724,E2 -6858.724} C_VEL
LIN {X 0,Y 481.658,Z 226.984,A -85,B 0,C 180,E1 -6861.397,E2 -6861.397} C_VEL
LIN {X 0,Y 481.661,Z 226.982,A -85,B 0,C 180,E1 -6864.116,E2 -6864.116} C_VEL
LIN {X 0,Y 481.667,Z 226.989,A -85,B 0,C 180,E1 -6867.119,E2 -6867.119} C_VEL
LIN {X 0,Y 481.679,Z 226.981,A -85,B 0,C 180,E1 -6869.743,E2 -6869.743} C_VEL
LIN {X 0,Y 481.665,Z 226.983,A -85,B 0,C 180,E1 -6872.677,E2 -6872.677} C_VEL
LIN {X 0,Y 481.642,Z 226.987,A -85,B 0,C 180,E1 -6875.711,E2 -6875.711} C_VEL
LIN {X 0,Y 481.68,Z 226.981,A -85,B 0,C 180,E1 -6878.861,E2 -6878.861} C_VEL
LIN {X 0,Y 481.63,Z 226.987,A -85,B 0,C 180,E1 -6882.165,E2 -6882.165} C_VEL
LIN {X 0,Y 481.668,Z 226.981,A -85,B 0,C 180,E1 -6884.459,E2 -6884.459} C_VEL
LIN {X 0,Y 481.629,Z 226.986,A -85,B 0,C 180,E1 -6886.856,E2 -6886.856} C_VEL
LIN {X 0,Y 481.671,Z 226.985,A -85,B 0,C 180,E1 -6890.058,E2 -6890.058} C_VEL
LIN {X 0,Y 481.633,Z 226.986,A -85,B 0,C 180,E1 -6893.252,E2 -6893.252} C_VEL
LIN {X 0,Y 481.708,Z 226.98,A -85,B 0,C 180,E1 -6896.329,E2 -6896.329} C_VEL
LIN {X 0,Y 481.661,Z 226.983,A -85,B 0,C 180,E1 -6899.418,E2 -6899.418} C_VEL
LIN {X 0,Y 481.681,Z 226.986,A -85,B 0,C 180,E1 -6902.166,E2 -6902.166} C_VEL
LIN {X 0,Y 481.727,Z 227.122,A -85,B 0,C 180,E1 -6905.545,E2 -6905.545} C_VEL
LIN {X 0,Y 483.494,Z 237.363,A -85,B 0,C 180,E1 -6907.568,E2 -6907.568} C_VEL
LIN {X 0,Y 482.868,Z 254.253,A -85,B 0,C 180,E1 -6910.647,E2 -6910.647} C_VEL
LIN {X 0,Y 482.338,Z 270.104,A -85,B 0,C 180,E1 -6913.472,E2 -6913.472} C_VEL
LIN {X 0,Y 482.802,Z 273.478,A -85,B 0,C 180,E1 -6913.591,E2 -6913.591} C_VEL
LIN {X 0,Y 484.843,Z 286.965,A -85,B 0,C 180,E1 -6913.863,E2 -6913.863} C_VEL
LIN {X 0,Y 484.216,Z 377.7,A -85,B 0,C 180,E1 -6915.231,E2 -6915.231} C_VEL
LIN {X 0,Y 483.89,Z 391.064,A -85,B 0,C 180,E1 -6915.597,E2 -6915.597} C_VEL
LIN {X 0,Y 483.516,Z 403.84,A -85,B 0,C 180,E1 -6916.122,E2 -6916.122} C_VEL
LIN {X 0,Y 483.144,Z 415.511,A -85,B 0,C 180,E1 -6916.776,E2 -6916.776} C_VEL
LIN {X 0,Y 482.735,Z 426.882,A -85,B 0,C 180,E1 -6917.598,E2 -6917.598} C_VEL
LIN {X 0,Y 482.286,Z 437.389,A -85,B 0,C 180,E1 -6918.547,E2 -6918.547} C_VEL
LIN {X 0,Y 481.866,Z 445.974,A -85,B 0,C 180,E1 -6919.494,E2 -6919.494} C_VEL
LIN {X 0,Y 481.535,Z 453.889,A -85,B 0,C 180,E1 -6920.548,E2 -6920.548} C_VEL
LIN {X 0,Y 481.26,Z 461.621,A -85,B 0,C 180,E1 -6921.813,E2 -6921.813} C_VEL
LIN {X 0,Y 481.02,Z 468.731,A -85,B 0,C 180,E1 -6923.286,E2 -6923.286} C_VEL
LIN {X 0,Y 480.963,Z 473.464,A -85,B 0,C 180,E1 -6924.549,E2 -6924.549} C_VEL
LIN {X 0,Y 480.831,Z 477.077,A -85,B 0,C 180,E1 -6925.808,E2 -6925.808} C_VEL
LIN {X 0,Y 480.873,Z 478.944,A -85,B 0,C 180,E1 -6926.647,E2 -6926.647} C_VEL
LIN {X 0,Y 480.792,Z 481.34,A -85,B 0,C 180,E1 -6928.323,E2 -6928.323} C_VEL
LIN {X 0,Y 480.745,Z 482.169,A -85,B 0,C 180,E1 -6929.999,E2 -6929.999} C_VEL
LIN {X 0,Y 480.762,Z 481.957,A -85,B 0,C 180,E1 -6930.836,E2 -6930.836} C_VEL
LIN {X 0,Y 480.791,Z 481.352,A -85,B 0,C 180,E1 -6931.674,E2 -6931.674} C_VEL
LIN {X 0,Y 480.872,Z 478.971,A -85,B 0,C 180,E1 -6933.35,E2 -6933.35} C_VEL
LIN {X 0,Y 480.841,Z 476.042,A -85,B 0,C 180,E1 -6934.61,E2 -6934.61} C_VEL
LIN {X 0,Y 480.962,Z 472.08,A -85,B 0,C 180,E1 -6935.869,E2 -6935.869} C_VEL
LIN {X 0,Y 481.111,Z 465.985,A -85,B 0,C 180,E1 -6937.342,E2 -6937.342} C_VEL
LIN {X 0,Y 481.357,Z 459.323,A -85,B 0,C 180,E1 -6938.605,E2 -6938.605} C_VEL
LIN {X 0,Y 481.693,Z 451.055,A -85,B 0,C 180,E1 -6939.87,E2 -6939.87} C_VEL
LIN {X 0,Y 482.02,Z 442.583,A -85,B 0,C 180,E1 -6940.925,E2 -6940.925} C_VEL
LIN {X 0,Y 482.567,Z 432.114,A -85,B 0,C 180,E1 -6941.976,E2 -6941.976} C_VEL
LIN {X 0,Y 482.97,Z 420.476,A -85,B 0,C 180,E1 -6942.916,E2 -6942.916} C_VEL
LIN {X 0,Y 483.385,Z 408.489,A -85,B 0,C 180,E1 -6943.664,E2 -6943.664} C_VEL
LIN {X 0,Y 483.865,Z 396.178,A -85,B 0,C 180,E1 -6944.24,E2 -6944.24} C_VEL
LIN {X 0,Y 484.18,Z 383.569,A -85,B 0,C 180,E1 -6944.66,E2 -6944.66} C_VEL
LIN {X 0,Y 484.401,Z 370.52,A -85,B 0,C 180,E1 -6944.922,E2 -6944.922} C_VEL
LIN {X 0,Y 484.858,Z 285.227,A -85,B 0,C 180,E1 -6946.206,E2 -6946.206} C_VEL
LIN {X 0,Y 482.387,Z 270.57,A -85,B 0,C 180,E1 -6946.533,E2 -6946.533} C_VEL
LIN {X 0,Y 482.362,Z 269.01,A -85,B 0,C 180,E1 -6946.722,E2 -6946.722} C_VEL
LIN {X 0,Y 482.95,Z 252.011,A -85,B 0,C 180,E1 -6949.774,E2 -6949.774} C_VEL
LIN {X 0,Y 483.557,Z 237.431,A -85,B 0,C 180,E1 -6952.426,E2 -6952.426} C_VEL
LIN {X 0,Y 481.722,Z 227.214,A -85,B 0,C 180,E1 -6954.453,E2 -6954.453} C_VEL
LIN {X 0,Y 481.718,Z 226.981,A -85,B 0,C 180,E1 -6957.13,E2 -6957.13} C_VEL
LIN {X 0,Y 481.68,Z 226.989,A -85,B 0,C 180,E1 -6959.739,E2 -6959.739} C_VEL
LIN {X 0,Y 481.674,Z 226.981,A -85,B 0,C 180,E1 -6962.672,E2 -6962.672} C_VEL
LIN {X 0,Y 481.633,Z 226.988,A -85,B 0,C 180,E1 -6965.708,E2 -6965.708} C_VEL
LIN {X 0,Y 481.668,Z 226.982,A -85,B 0,C 180,E1 -6968.857,E2 -6968.857} C_VEL
LIN {X 0,Y 481.646,Z 226.986,A -85,B 0,C 180,E1 -6971.91,E2 -6971.91} C_VEL
LIN {X 0,Y 481.653,Z 226.989,A -85,B 0,C 180,E1 -6974.456,E2 -6974.456} C_VEL
LIN {X 0,Y 481.639,Z 226.982,A -85,B 0,C 180,E1 -6977.836,E2 -6977.836} C_VEL
LIN {X 0,Y 481.663,Z 226.983,A -85,B 0,C 180,E1 -6981.138,E2 -6981.138} C_VEL
LIN {X 0,Y 481.657,Z 226.989,A -85,B 0,C 180,E1 -6984.794,E2 -6984.794} C_VEL
LIN {X 0,Y 481.668,Z 226.98,A -85,B 0,C 180,E1 -6987.323,E2 -6987.323} C_VEL
LIN {X 0,Y 481.667,Z 226.985,A -85,B 0,C 180,E1 -6990.256,E2 -6990.256} C_VEL
LIN {X 0,Y 481.657,Z 226.986,A -85,B 0,C 180,E1 -6993.104,E2 -6993.104} C_VEL
LIN {X 0,Y 481.641,Z 226.984,A -85,B 0,C 180,E1 -6995.882,E2 -6995.882} C_VEL
LIN {X 0,Y 481.696,Z 226.982,A -85,B 0,C 180,E1 -6999.025,E2 -6999.025} C_VEL
LIN {X 0,Y 481.679,Z 226.979,A -85,B 0,C 180,E1 -7002.155,E2 -7002.155} C_VEL
LIN {X 0,Y 481.729,Z 226.976,A -85,B 0,C 180,E1 -7004.773,E2 -7004.773} C_VEL
LIN {X 0,Y 481.739,Z 226.969,A -85,B 0,C 180,E1 -7008.212,E2 -7008.212} C_VEL
LIN {X 0,Y 481.707,Z 226.976,A -85,B 0,C 180,E1 -7011.608,E2 -7011.608} C_VEL
LIN {X 0,Y 481.78,Z 226.968,A -85,B 0,C 180,E1 -7014.136,E2 -7014.136} C_VEL
LIN {X 0,Y 481.89,Z 226.958,A -85,B 0,C 180,E1 -7017.489,E2 -7017.489} C_VEL
LIN {X 0,Y 481.89,Z 226.955,A -85,B 0,C 180,E1 -7019.997,E2 -7019.997} C_VEL
LIN {X 0,Y 481.89,Z 226.953,A -85,B 0,C 180,E1 -7022.504,E2 -7022.504} C_VEL
LIN {X 0,Y 481.754,Z 226.976,A -85,B 0,C 180,E1 -7025.858,E2 -7025.858} C_VEL
LIN {X 0,Y 481.716,Z 226.976,A -85,B 0,C 180,E1 -7028.386,E2 -7028.386} C_VEL
LIN {X 0,Y 481.73,Z 226.982,A -85,B 0,C 180,E1 -7031.782,E2 -7031.782} C_VEL
LIN {X 0,Y 481.716,Z 226.977,A -85,B 0,C 180,E1 -7035.221,E2 -7035.221} C_VEL
LIN {X 0,Y 481.682,Z 226.981,A -85,B 0,C 180,E1 -7038.719,E2 -7038.719} C_VEL
LIN {X 0,Y 481.619,Z 226.989,A -85,B 0,C 180,E1 -7041.392,E2 -7041.392} C_VEL
LIN {X 0,Y 481.631,Z 226.994,A -85,B 0,C 180,E1 -7044.111,E2 -7044.111} C_VEL
LIN {X 0,Y 481.717,Z 226.976,A -85,B 0,C 180,E1 -7047.136,E2 -7047.136} C_VEL
LIN {X 0,Y 481.648,Z 226.983,A -85,B 0,C 180,E1 -7049.738,E2 -7049.738} C_VEL
LIN {X 0,Y 481.64,Z 226.988,A -85,B 0,C 180,E1 -7052.671,E2 -7052.671} C_VEL
LIN {X 0,Y 481.61,Z 226.987,A -85,B 0,C 180,E1 -7055.706,E2 -7055.706} C_VEL
LIN {X 0,Y 481.685,Z 226.983,A -85,B 0,C 180,E1 -7059.352,E2 -7059.352} C_VEL
LIN {X 0,Y 481.639,Z 226.99,A -85,B 0,C 180,E1 -7062.155,E2 -7062.155} C_VEL
LIN {X 0,Y 481.622,Z 226.994,A -85,B 0,C 180,E1 -7064.455,E2 -7064.455} C_VEL
LIN {X 0,Y 481.644,Z 227.073,A -85,B 0,C 180,E1 -7066.631,E2 -7066.631} C_VEL
LIN {X 0,Y 482.872,Z 233.48,A -85,B 0,C 180,E1 -7067.973,E2 -7067.973} C_VEL
LIN {X 0,Y 482.746,Z 243.614,A -85,B 0,C 180,E1 -7069.896,E2 -7069.896} C_VEL
LIN {X 0,Y 482.378,Z 257.646,A -85,B 0,C 180,E1 -7072.482,E2 -7072.482} C_VEL
LIN {X 0,Y 483.403,Z 263.461,A -85,B 0,C 180,E1 -7072.647,E2 -7072.647} C_VEL
LIN {X 0,Y 484.989,Z 273.481,A -85,B 0,C 180,E1 -7072.86,E2 -7072.86} C_VEL
LIN {X 0,Y 484.282,Z 365.305,A -85,B 0,C 180,E1 -7074.257,E2 -7074.257} C_VEL
LIN {X 0,Y 484.125,Z 375.037,A -85,B 0,C 180,E1 -7074.512,E2 -7074.512} C_VEL
LIN {X 0,Y 483.444,Z 380.731,A -85,B 0,C 180,E1 -7074.681,E2 -7074.681} C_VEL
LIN {X 0,Y 480.406,Z 389.844,A -85,B 0,C 180,E1 -7074.977,E2 -7074.977} C_VEL
LIN {X 0,Y 477.233,Z 398.656,A -85,B 0,C 180,E1 -7075.367,E2 -7075.367} C_VEL
LIN {X 0,Y 476.347,Z 403.878,A -85,B 0,C 180,E1 -7075.681,E2 -7075.681} C_VEL
LIN {X 0,Y 475.844,Z 414.748,A -85,B 0,C 180,E1 -7076.497,E2 -7076.497} C_VEL
LIN {X 0,Y 475.382,Z 424.621,A -85,B 0,C 180,E1 -7077.415,E2 -7077.415} C_VEL
LIN {X 0,Y 475.035,Z 432.64,A -85,B 0,C 180,E1 -7078.319,E2 -7078.319} C_VEL
LIN {X 0,Y 474.627,Z 441.77,A -85,B 0,C 180,E1 -7079.571,E2 -7079.571} C_VEL
LIN {X 0,Y 474.315,Z 449.717,A -85,B 0,C 180,E1 -7080.941,E2 -7080.941} C_VEL
LIN {X 0,Y 474.056,Z 455.403,A -85,B 0,C 180,E1 -7082.162,E2 -7082.162} C_VEL
LIN {X 0,Y 473.887,Z 460.615,A -85,B 0,C 180,E1 -7083.584,E2 -7083.584} C_VEL
LIN {X 0,Y 473.774,Z 463.961,A -85,B 0,C 180,E1 -7084.794,E2 -7084.794} C_VEL
LIN {X 0,Y 473.593,Z 467.023,A -85,B 0,C 180,E1 -7086.381,E2 -7086.381} C_VEL
LIN {X 0,Y 473.58,Z 468.114,A -85,B 0,C 180,E1 -7087.306,E2 -7087.306} C_VEL
LIN {X 0,Y 473.566,Z 468.761,A -85,B 0,C 180,E1 -7088.223,E2 -7088.223} C_VEL
LIN {X 0,Y 473.602,Z 468.925,A -85,B 0,C 180,E1 -7089.194,E2 -7089.194} C_VEL
LIN {X 0,Y 473.611,Z 468.64,A -85,B 0,C 180,E1 -7090.045,E2 -7090.045} C_VEL
LIN {X 0,Y 473.649,Z 466.953,A -85,B 0,C 180,E1 -7091.72,E2 -7091.72} C_VEL
LIN {X 0,Y 473.711,Z 464.144,A -85,B 0,C 180,E1 -7093.185,E2 -7093.185} C_VEL
LIN {X 0,Y 473.874,Z 460.308,A -85,B 0,C 180,E1 -7094.561,E2 -7094.561} C_VEL
LIN {X 0,Y 474.015,Z 455.608,A -85,B 0,C 180,E1 -7095.841,E2 -7095.841} C_VEL
LIN {X 0,Y 474.226,Z 449.473,A -85,B 0,C 180,E1 -7097.157,E2 -7097.157} C_VEL
LIN {X 0,Y 474.555,Z 441.832,A -85,B 0,C 180,E1 -7098.469,E2 -7098.469} C_VEL
LIN {X 0,Y 474.914,Z 434.031,A -85,B 0,C 180,E1 -7099.557,E2 -7099.557} C_VEL
LIN {X 0,Y 475.343,Z 424.523,A -85,B 0,C 180,E1 -7100.641,E2 -7100.641} C_VEL
LIN {X 0,Y 475.866,Z 413.422,A -85,B 0,C 180,E1 -7101.657,E2 -7101.657} C_VEL
LIN {X 0,Y 476.357,Z 402.155,A -85,B 0,C 180,E1 -7102.478,E2 -7102.478} C_VEL
LIN {X 0,Y 476.79,Z 390.694,A -85,B 0,C 180,E1 -7103.123,E2 -7103.123} C_VEL
LIN {X 0,Y 477.114,Z 377.846,A -85,B 0,C 180,E1 -7103.659,E2 -7103.659} C_VEL
LIN {X 0,Y 477.39,Z 365.405,A -85,B 0,C 180,E1 -7104.007,E2 -7104.007} C_VEL
LIN {X 0,Y 477.911,Z 272.418,A -85,B 0,C 180,E1 -7105.441,E2 -7105.441} C_VEL
LIN {X 0,Y 475.405,Z 258.406,A -85,B 0,C 180,E1 -7105.762,E2 -7105.762} C_VEL
LIN {X 0,Y 475.377,Z 257.393,A -85,B 0,C 180,E1 -7105.868,E2 -7105.868} C_VEL
LIN {X 0,Y 475.964,Z 242.826,A -85,B 0,C 180,E1 -7108.732,E2 -7108.732} C_VEL
LIN {X 0,Y 476.061,Z 235.442,A -85,B 0,C 180,E1 -7110.213,E2 -7110.213} C_VEL
LIN {X 0,Y 474.766,Z 227.91,A -85,B 0,C 180,E1 -7111.857,E2 -7111.857} C_VEL
LIN {X 0,Y 474.645,Z 227.864,A -85,B 0,C 180,E1 -7113.397,E2 -7113.397} C_VEL
LIN {X 0,Y 474.732,Z 227.85,A -85,B 0,C 180,E1 -7115.949,E2 -7115.949} C_VEL
LIN {X 0,Y 474.685,Z 227.851,A -85,B 0,C 180,E1 -7118.516,E2 -7118.516} C_VEL
LIN {X 0,Y 474.697,Z 227.853,A -85,B 0,C 180,E1 -7121.964,E2 -7121.964} C_VEL
LIN {X 0,Y 474.64,Z 227.865,A -85,B 0,C 180,E1 -7125.77,E2 -7125.77} C_VEL
LIN {X 0,Y 474.626,Z 227.858,A -85,B 0,C 180,E1 -7129.013,E2 -7129.013} C_VEL
LIN {X 0,Y 474.55,Z 227.873,A -85,B 0,C 180,E1 -7131.732,E2 -7131.732} C_VEL
LIN {X 0,Y 474.593,Z 227.865,A -85,B 0,C 180,E1 -7134.498,E2 -7134.498} C_VEL
LIN {X 0,Y 474.602,Z 227.861,A -85,B 0,C 180,E1 -7137.327,E2 -7137.327} C_VEL
LIN {X 0,Y 474.569,Z 227.874,A -85,B 0,C 180,E1 -7140.234,E2 -7140.234} C_VEL
LIN {X 0,Y 474.583,Z 227.863,A -85,B 0,C 180,E1 -7143.226,E2 -7143.226} C_VEL
LIN {X 0,Y 474.548,Z 227.876,A -85,B 0,C 180,E1 -7146.328,E2 -7146.328} C_VEL
LIN {X 0,Y 474.572,Z 227.865,A -85,B 0,C 180,E1 -7149.647,E2 -7149.647} C_VEL
LIN {X 0,Y 474.548,Z 227.872,A -85,B 0,C 180,E1 -7152.943,E2 -7152.943} C_VEL
LIN {X 0,Y 474.579,Z 227.864,A -85,B 0,C 180,E1 -7155.898,E2 -7155.898} C_VEL
LIN {X 0,Y 474.584,Z 227.869,A -85,B 0,C 180,E1 -7159.048,E2 -7159.048} C_VEL
LIN {X 0,Y 474.589,Z 227.863,A -85,B 0,C 180,E1 -7161.709,E2 -7161.709} C_VEL
LIN {X 0,Y 474.606,Z 227.865,A -85,B 0,C 180,E1 -7164.73,E2 -7164.73} C_VEL
LIN {X 0,Y 474.612,Z 227.861,A -85,B 0,C 180,E1 -7167.791,E2 -7167.791} C_VEL
LIN {X 0,Y 474.586,Z 227.867,A -85,B 0,C 180,E1 -7170.895,E2 -7170.895} C_VEL
LIN {X 0,Y 474.57,Z 227.869,A -85,B 0,C 180,E1 -7173.628,E2 -7173.628} C_VEL
LIN {X 0,Y 474.627,Z 227.858,A -85,B 0,C 180,E1 -7176.646,E2 -7176.646} C_VEL
LIN {X 0,Y 474.646,Z 227.857,A -85,B 0,C 180,E1 -7180.094,E2 -7180.094} C_VEL
LIN {X 0,Y 474.623,Z 227.859,A -85,B 0,C 180,E1 -7182.778,E2 -7182.778} C_VEL
LIN {X 0,Y 474.638,Z 227.862,A -85,B 0,C 180,E1 -7185.425,E2 -7185.425} C_VEL
LIN {X 0,Y 474.692,Z 227.855,A -85,B 0,C 180,E1 -7188.041,E2 -7188.041} C_VEL
LIN {X 0,Y 474.67,Z 227.856,A -85,B 0,C 180,E1 -7191.489,E2 -7191.489} C_VEL
LIN {X 0,Y 474.738,Z 227.852,A -85,B 0,C 180,E1 -7194.055,E2 -7194.055} C_VEL
LIN {X 0,Y 474.876,Z 227.828,A -85,B 0,C 180,E1 -7197.459,E2 -7197.459} C_VEL
LIN {X 0,Y 474.884,Z 227.833,A -85,B 0,C 180,E1 -7200.003,E2 -7200.003} C_VEL
LIN {X 0,Y 474.877,Z 227.831,A -85,B 0,C 180,E1 -7202.548,E2 -7202.548} C_VEL
LIN {X 0,Y 474.745,Z 227.846,A -85,B 0,C 180,E1 -7205.951,E2 -7205.951} C_VEL
LIN {X 0,Y 474.675,Z 227.86,A -85,B 0,C 180,E1 -7208.517,E2 -7208.517} C_VEL
LIN {X 0,Y 474.715,Z 227.848,A -85,B 0,C 180,E1 -7211.965,E2 -7211.965} C_VEL
LIN {X 0,Y 474.692,Z 227.85,A -85,B 0,C 180,E1 -7215.769,E2 -7215.769} C_VEL
LIN {X 0,Y 474.673,Z 227.858,A -85,B 0,C 180,E1 -7219.013,E2 -7219.013} C_VEL
LIN {X 0,Y 474.6,Z 227.861,A -85,B 0,C 180,E1 -7221.731,E2 -7221.731} C_VEL
LIN {X 0,Y 474.639,Z 227.859,A -85,B 0,C 180,E1 -7224.497,E2 -7224.497} C_VEL
LIN {X 0,Y 474.613,Z 227.864,A -85,B 0,C 180,E1 -7227.328,E2 -7227.328} C_VEL
LIN {X 0,Y 474.609,Z 227.86,A -85,B 0,C 180,E1 -7230.232,E2 -7230.232} C_VEL
LIN {X 0,Y 474.629,Z 227.867,A -85,B 0,C 180,E1 -7233.224,E2 -7233.224} C_VEL
LIN {X 0,Y 474.596,Z 227.862,A -85,B 0,C 180,E1 -7236.325,E2 -7236.325} C_VEL
LIN {X 0,Y 474.637,Z 227.864,A -85,B 0,C 180,E1 -7239.549,E2 -7239.549} C_VEL
LIN {X 0,Y 474.59,Z 227.863,A -85,B 0,C 180,E1 -7242.231,E2 -7242.231} C_VEL
LIN {X 0,Y 474.63,Z 227.862,A -85,B 0,C 180,E1 -7245.298,E2 -7245.298} C_VEL
LIN {X 0,Y 474.606,Z 227.863,A -85,B 0,C 180,E1 -7248.212,E2 -7248.212} C_VEL
LIN {X 0,Y 474.621,Z 227.863,A -85,B 0,C 180,E1 -7251.542,E2 -7251.542} C_VEL
LIN {X 0,Y 474.635,Z 227.857,A -85,B 0,C 180,E1 -7254.725,E2 -7254.725} C_VEL
LIN {X 0,Y 474.648,Z 227.86,A -85,B 0,C 180,E1 -7257.787,E2 -7257.787} C_VEL
LIN {X 0,Y 474.62,Z 227.863,A -85,B 0,C 180,E1 -7260.888,E2 -7260.888} C_VEL
LIN {X 0,Y 474.625,Z 227.864,A -85,B 0,C 180,E1 -7263.625,E2 -7263.625} C_VEL
LIN {X 0,Y 474.676,Z 228.07,A -85,B 0,C 180,E1 -7265.39,E2 -7265.39} C_VEL
LIN {X 0,Y 476.521,Z 238.404,A -85,B 0,C 180,E1 -7267.45,E2 -7267.45} C_VEL
LIN {X 0,Y 475.929,Z 254.304,A -85,B 0,C 180,E1 -7270.391,E2 -7270.391} C_VEL
LIN {X 0,Y 475.362,Z 270.147,A -85,B 0,C 180,E1 -7273.244,E2 -7273.244} C_VEL
LIN {X 0,Y 476.103,Z 275.118,A -85,B 0,C 180,E1 -7273.389,E2 -7273.389} C_VEL
LIN {X 0,Y 478.014,Z 287.058,A -85,B 0,C 180,E1 -7273.638,E2 -7273.638} C_VEL
LIN {X 0,Y 477.346,Z 378.459,A -85,B 0,C 180,E1 -7275.041,E2 -7275.041} C_VEL
LIN {X 0,Y 476.984,Z 392.291,A -85,B 0,C 180,E1 -7275.438,E2 -7275.438} C_VEL
LIN {X 0,Y 476.559,Z 404.699,A -85,B 0,C 180,E1 -7275.97,E2 -7275.97} C_VEL
LIN {X 0,Y 476.158,Z 416.582,A -85,B 0,C 180,E1 -7276.665,E2 -7276.665} C_VEL
LIN {X 0,Y 475.738,Z 428.149,A -85,B 0,C 180,E1 -7277.534,E2 -7277.534} C_VEL
LIN {X 0,Y 475.246,Z 438.286,A -85,B 0,C 180,E1 -7278.483,E2 -7278.483} C_VEL
LIN {X 0,Y 474.786,Z 447.522,A -85,B 0,C 180,E1 -7279.552,E2 -7279.552} C_VEL
LIN {X 0,Y 474.375,Z 456.5,A -85,B 0,C 180,E1 -7280.835,E2 -7280.835} C_VEL
LIN {X 0,Y 474.113,Z 463.729,A -85,B 0,C 180,E1 -7282.118,E2 -7282.118} C_VEL
LIN {X 0,Y 473.907,Z 469.981,A -85,B 0,C 180,E1 -7283.526,E2 -7283.526} C_VEL
LIN {X 0,Y 473.839,Z 474.664,A -85,B 0,C 180,E1 -7284.893,E2 -7284.893} C_VEL
LIN {X 0,Y 473.737,Z 476.964,A -85,B 0,C 180,E1 -7285.745,E2 -7285.745} C_VEL
LIN {X 0,Y 473.768,Z 478.835,A -85,B 0,C 180,E1 -7286.597,E2 -7286.597} C_VEL
LIN {X 0,Y 473.725,Z 480.237,A -85,B 0,C 180,E1 -7287.448,E2 -7287.448} C_VEL
LIN {X 0,Y 473.69,Z 481.848,A -85,B 0,C 180,E1 -7289.149,E2 -7289.149} C_VEL
LIN {X 0,Y 473.672,Z 482.071,A -85,B 0,C 180,E1 -7289.999,E2 -7289.999} C_VEL
LIN {X 0,Y 473.69,Z 481.861,A -85,B 0,C 180,E1 -7290.849,E2 -7290.849} C_VEL
LIN {X 0,Y 473.725,Z 480.268,A -85,B 0,C 180,E1 -7292.55,E2 -7292.55} C_VEL
LIN {X 0,Y 473.767,Z 478.88,A -85,B 0,C 180,E1 -7293.4,E2 -7293.4} C_VEL
